Staubli VAL3: TEACH.pjx

--- TEACH.pjx ---
Parameters version=s7.7.1 stackSize=5000 millimeterUnit=true
Program file=AdjustTraj.pgx
Program file=Approach.pgx
Program file=Cut.pgx
Program file=GetListItems.pgx
Program file=GetProductMess.pgx
Program file=IdlePoint.pgx
Program file=IsPointOK.pgx
Program file=Leave.pgx
Program file=OnAction.pgx
Program file=OneWpMproChoose.pgx
Program file=Product.pgx
Program file=SetTrajPara.pgx
Program file=Simulate.pgx
Program file=SingleMove.pgx
Program file=start.pgx
Program file=stop.pgx
Program file=Teach2Tool.pgx
Program file=TeachAction.pgx
Program file=TeachAxis.pgx
Program file=TeachConfig.pgx
Program file=TeachFrame.pgx
Program file=TeachHome.pgx
Program file=TeachNewTraj.pgx
Program file=TeachOffset.pgx
Program file=TeachPreset.pgx
Program file=TeachProduct.pgx
Program file=TeachRecipe.pgx
Program file=TeachRemote.pgx
Program file=TeachSyncAxis.pgx
Program file=TeachTool.pgx
Program file=TrajScreen.pgx
Program file=WeldTraj.pgx
Program file=WorkPlaceChose.pgx
Data file=Teach.dtx
Library alias=TxtFile path=Disk://TxtFile/TxtFile.pjx
Library alias=DataBase path=Disk://DataBase/DataBase.pjx
Library alias=Kit path=Disk://Kit/Kit.pjx
Library alias=UI path=Disk://StaubliUI/StaubliUI.pjx
Library alias=Motion path=Disk://Motion/Motion.pjx
Library alias=IO path=Disk://IO/IO.pjx
Library alias=Algorith path=Disk://Algorith/Algorith.pjx
Library alias=CalTool path=Disk://StaubliCalTool7/StaubliCalTool7.pjx
Library alias=ExtAxis path=Disk://extAxisCan/extAxisCan.pjx autoload=false
Library alias=Custom path=Disk://Custom/Custom.pjx

--- TEACH.dtx ---
mdesc mNomSpeed
num nApproIndex
num nCutIndex
num nLeaveIndex
public num nPointType
string sSItem
public num nTrajIndex
public string sMess
num nCutMc
bool bPowerFlag
bool bFirstTeach
num nTeachAction
bool bSyc
public num n500Count
num nPartID
bool bSaveTxt
bool bCheckAxisSafte
num nCursonIndex
num nAxisSpeed

--- start.pgx ---
public program start()
begin














end

--- AdjustTraj.pgx ---
public program AdjustTraj(num x_nTrajIndex)
  local bool l_bRes
  local num l_nNum
begin


  //调图主界面，入口

  cls()

  call UI:Control_PanelMd("请等待，正在读取文件......")
  TxtFile:bStartRead=true
  DataBase:bStopPoll=true

  //删除临时文件
  if $fileExists("Disk://Txt/1.txt")
    $delete("Disk://Txt/1.txt")
  endIf

  if $fileExists("Disk://Txt/2.txt")
    $delete("Disk://Txt/2.txt")
  endIf

  if $fileExists("Disk://Txt/3.txt")
    $delete("Disk://Txt/3.txt")
  endIf

  if $fileExists("Disk://Txt/4.txt")
    $delete("Disk://Txt/4.txt")
  endIf




  call TxtFile:IsAdjustTraj("Disk://Txt/Recipe.txt",TxtFile:sProductName,x_nTrajIndex,x_nTrajIndex,l_bRes)
  call TxtFile:CloseFile()
  if !l_bRes
    DataBase:bStopPoll=false
    popUpMsg("文件读取出错!")
    return
  endIf


  //参数初始化
  bFirstTeach=true
  DataBase:bStopPoll=false
  //路径界面
  call TrajScreen()


end

--- APPROACH.pgx ---
public program Approach()
  local num l_nKey
  local bool l_bRes
  local string l_sProductName
  local jointRx l_jBuff
  local bool l_bCut
  local bool l_bMoveL
  local bool l_bFirst
  local trsf l_trTrsf
  local num l_nNum
  local num l_nAtPosition
begin
  //趋近点主界面
  //  $jogContext(TxtFile:tCfg,TxtFile:fArray,0)








  TxtFile:fArray.trsf={0,0,0,0,0,0}

  //2014.2.17  在哪个坐标系中运动
  if !DataBase:bWorldMove
    $jogContext(TxtFile:tCfg,TxtFile:fArray,0)
  else
    $jogContext(TxtFile:tCfg,world,0)
  endIf


  call IO:KeyDigtalIO(false,false,false,0,0)

  TxtFile:fArray.trsf={0,0,0,0,0,0}
  cls()
  while  nPointType==1
    l_nKey=getKey()
    switch l_nKey
      //上移
      case 261
        nApproIndex=max(nApproIndex-1,0)


      break

      //下移
      case 266
        nApproIndex=min(nApproIndex+1,size(TxtFile:pAppro)-1)

      break


      //向右
      //2015.08.10
      case 268
        nPointType=2
      break


      //插入
      case 271

        insert(TxtFile:pAppro[nApproIndex+1])
        insert(TxtFile:jAppro[nApproIndex+1])
        insert(TxtFile:bAppro[nApproIndex+1])
        insert(TxtFile:trAppro[nApproIndex+1])
        //外部轴
        insert(TxtFile:trApproAxis[nApproIndex+1])
        TxtFile:pAppro[nApproIndex+1]=TxtFile:pAppro[nApproIndex]
        TxtFile:jAppro[nApproIndex+1]=TxtFile:jAppro[nApproIndex]
        TxtFile:bAppro[nApproIndex+1]=TxtFile:bAppro[nApproIndex]
        TxtFile:trAppro[nApproIndex+1]=TxtFile:trAppro[nApproIndex]
        //外部轴
        TxtFile:trApproAxis[nApproIndex+1]=TxtFile:trApproAxis[nApproIndex]


        nApproIndex=nApproIndex+1
        TxtFile:trPointCount.x=size(TxtFile:pAppro)

        //2014.5.30
        //××××××××××××××××××××××
        if TxtFile:nSingleType!=20 and TxtFile:nSingleType!=9
          TxtFile:pAppro[nApproIndex]=here(TxtFile:tCfg,TxtFile:fArray)
          if TxtFile:fPofffset.trsf=={0,0,0,0,0,0} and TxtFile:fToffset.trsf=={0,0,0,0,0,0} and TxtFile:fArray.trsf=={0,0,0,0,0,0}
            TxtFile:jAppro[nApproIndex]=herej()
          else
            call Motion:Point2Joint(TxtFile:pAppro[nApproIndex], TxtFile:jAppro[nApproIndex],l_bRes)
            if !l_bRes
              popUpMsg("Joint数据转换出错")
            endIf
          endIf
        endIf

        //××××××××××××××××××××××××




      break


      //记录
      case 272
        TxtFile:fArray.trsf={0,0,0,0,0,0}
        //2015.08.10
        l_bRes=true
        //call UI:Control_YesNO("确定要记录吗?",l_bRes)

        if l_bRes
          TxtFile:pAppro[nApproIndex]=here(TxtFile:tCfg,TxtFile:fArray)
          if TxtFile:fPofffset.trsf=={0,0,0,0,0,0} and TxtFile:fToffset.trsf=={0,0,0,0,0,0} and TxtFile:fArray.trsf=={0,0,0,0,0,0}
            TxtFile:jAppro[nApproIndex]=herej()
          else
            call Motion:Point2Joint(TxtFile:pAppro[nApproIndex], TxtFile:jAppro[nApproIndex],l_bRes)
            if !l_bRes
              popUpMsg("Joint数据转换出错")
            endIf
          endIf

          //2014.07.28记录同步外部轴
          if TxtFile:nSingleType==20 or TxtFile:nSingleType==9
            call ExtAxis:RecordExtAxis(TxtFile:trApproAxis[nApproIndex],TxtFile:pAppro[nApproIndex].trsf,TxtFile:tCfg)
          endIf


        endIf
      break

      //参数
      case 273
        l_bMoveL=TxtFile:bAppro[nApproIndex]
        // call UI:Control_Para(TxtFile:trAppro[nApproIndex],TxtFile:bAppro[nApproIndex],false,0)
        call UI:Control_Para(TxtFile:trAppro,TxtFile:bAppro,false,TxtFile:nSingleType,nApproIndex,TxtFile:trApproAxis)
        //改变标志符
        if l_bMoveL!=TxtFile:bAppro[nApproIndex]
          //MOVEL
          if TxtFile:bAppro[nApproIndex]
            call Motion:Joint2Point(TxtFile:jAppro[nApproIndex],TxtFile:pAppro[nApproIndex])
          else
            //MOVEJ
            call Motion:Point2Joint(TxtFile:pAppro[nApproIndex], TxtFile:jAppro[nApproIndex],l_bRes)
            if !l_bRes
              popUpMsg("Joint数据转换出错")
            endIf
          endIf

          //2014.12.05记录同步外部轴
          if TxtFile:nSingleType==20 or TxtFile:nSingleType==9
            call ExtAxis:RecordExtAxis(TxtFile:trApproAxis[nApproIndex],TxtFile:pAppro[nApproIndex].trsf,TxtFile:tCfg)
          endIf


        endIf
      break

      //删除
      case 274
        if size(TxtFile:pAppro)==1
          popUpMsg("趋近点必须有一个")
        else
          call UI:Control_YesNO("确定要删除吗?",l_bRes)
          if l_bRes
            delete(TxtFile:pAppro[nApproIndex])
            delete(TxtFile:jAppro[nApproIndex])
            delete(TxtFile:bAppro[nApproIndex])
            delete(TxtFile:trAppro[nApproIndex])
            delete(TxtFile:trApproAxis[nApproIndex])
          endIf
        endIf
        TxtFile:trPointCount.x=size(TxtFile:pAppro)
      break


      //配置
      case 112,275
        call SetTrajPara()


      break

      //退出
      case 277
        call UI:Control_YesNO("确定要退出吗?",l_bRes)
        if l_bRes
          nPointType=-1
          return
        endIf
      break

      //上传
      case 278
        nPointType=2
      break

      //点位
      case 270
        if TxtFile:bAppro[nApproIndex]
          call UI:Control_Point(TxtFile:pAppro[nApproIndex] )
        else
          call UI:Control_Joint(TxtFile:jAppro[nApproIndex])
        endIf
        cls()
      break

      //****************************************
      //V
      //2014.12.02
      //外部PLC控制第七轴
      case 118
        if DataBase:bExtraContrAxis
          call UI:Control_YesNO("确定移动外部第七轴吗？",l_bRes)
          if l_bRes
            call UI:Control_PanelMd("外部第七轴正在运动....")
            resetMotion()
            call IO:ExtraContrAxis(TxtFile:trWorkplace.x,l_bRes)
            if !l_bRes
              popUpMsg("PLC控制外部轴数据错误,检查第七轴数据!")
              disablePower()
            endIf
          endIf
          cls()
        endIf
      break
      //******************************************




    endSwitch





    if (l_nKey<279  and l_nKey>=260)or l_nKey==112 or !l_bFirst or l_nKey==118
      l_bFirst=true
      call GetListItems()
      call UI:Form_PanelList("LasMAN3.6->示教路径","趋近点",sSItem,nApproIndex,"插入,记录,参数,删除,全局,,退出,继续")
      call UI:Control_Mess("类型:"+TxtFile:sTrajType[TxtFile:nSingleType],"趋近点个数:"+toString("",size(TxtFile:pAppro)))
      call SingleMove(1)



    endIf
    //2014.07.30
    //同步七八轴
    if (TxtFile:nSingleType==20 or TxtFile:nSingleType==9) and (TxtFile:bSync7Axis or TxtFile:bSync8Axis)
      call ExtAxis:RecordExtAxis(l_trTrsf,l_trTrsf,TxtFile:tCfg)

      gotoxy(1,12)
      put("七轴:"+toString(".3",l_trTrsf.x))
      if TxtFile:bSync8Axis
        gotoxy(20,12)
        put("八轴:"+toString(".3",l_trTrsf.y))
      endIf
    endIf
    //

    //为了表示到达位置
    //2015.08.10
    //2015.09.22
    //为整个列表进行修改

    if nApproIndex>10
      l_nAtPosition=nApproIndex-10
    else
      l_nAtPosition=0
    endIf

    for l_nNum=0 to min(size(TxtFile:bAppro)-1,10)
      gotoxy(22,min(l_nNum+1,10))
      setTextMode(sel((l_nAtPosition+l_nNum)==nApproIndex,1,0))


      if TxtFile:bAppro[l_nAtPosition+l_nNum]
        if distance(TxtFile:pAppro[l_nAtPosition+l_nNum],here(TxtFile:tFileTool,TxtFile:fArray))<0.1
          put("@")
        else
          put("│")
        endIf

      else
        if distance(jointToPoint(TxtFile:tFileTool,TxtFile:fArray,herej()),jointToPoint(TxtFile:tFileTool,TxtFile:fArray,TxtFile:jAppro[l_nAtPosition+l_nNum]))<0.1
          put("@")
        else
          put("│")
        endIf
      endIf
    endFor

    //*************************

    delay(0)

  endWhile



end

--- CUT.pgx ---
public program Cut()
  local num l_nKey
  local bool l_bRes
  local string l_sProductName
  local string l_sBottom
  local bool l_bCut
  local num l_nSaveTime
  local frame l_trOffset
  local num l_nTo[5]
  local num l_nFrom[5]
  local num l_nNum
  local bool l_bFirst
  local num l_nSpeed[2]
  local string l_sTtile
  local bool l_bBatPara[5]
  local num l_nBatPara[5]
  local num l_nFromTo[2]
  local trsf l_trTrsf
  local num l_nAtPosition
begin
  //切割点主界面
  //参数初始化
  // call IO:Follow(false)
  call IO:SafteyIO()
  TxtFile:fArray.trsf={0,0,0,0,0,0}


  //2014.2.17  在哪个坐标系中运动
  if !DataBase:bWorldMove
    $jogContext(TxtFile:tCfg,TxtFile:fArray,0)
  else
    $jogContext(TxtFile:tCfg,world,0)
  endIf

  //2014.2.18 区分焊接与切割
  if TxtFile:bWeldEnable
    l_sTtile="焊接点"
  else
    l_sTtile="切割点"
  endIf



  nPartID=1
  if TxtFile:trPointCount.y>500
    DataBase:bStopPoll=true
    call TxtFile:ReadPartTraj(nPartID,l_bRes)
  endIf
  DataBase:bStopPoll=false
  nCutMc=0
  l_nSaveTime=0
  n500Count=0

  if TxtFile:nSingleType!=10 and TxtFile:nSingleType!=20 and TxtFile:nSingleType!=9

    for l_nKey=0 to size(TxtFile:pCut)-1
      TxtFile:bMoveC[l_nKey]=false
    endFor
  endIf

  //界面
  call GetListItems()
  if TxtFile:nSingleType==10 or TxtFile:nSingleType==20
    l_sBottom="插入,记录,参数,删除,全局,偏差,返回,继续"
  else
    l_sBottom=",记录,参数,,全局,偏差,返回,继续"
  endIf


  //界面初始化
  resetMotion()
  cls()


  //循环
  while  nPointType==2
    DataBase:bStopPoll=false
    TxtFile:fArray.trsf={0,0,0,0,0,0}
    l_nKey=getKey()
    switch l_nKey

      //配置
      case 112,275
        call SetTrajPara()


      break

      //步进打开
      case 122
        //Z
        // if TxtFile:bStepMove
        TxtFile:nStepLength=max(0,TxtFile:nStepLength)
        call UI:Control_YesNO("确定使用步进"+toString(".1",TxtFile:nStepLength)+"毫米模式吗?",l_bRes)
        if l_bRes
          TxtFile:fArray.trsf={0,0,0,0,0,0}
          $jogContext(TxtFile:tCfg,TxtFile:fArray,TxtFile:nStepLength)
        endIf
        //  endIf
      break


      //步进关
      case 90

        TxtFile:fArray.trsf={0,0,0,0,0,0}
        $jogContext(TxtFile:tCfg,TxtFile:fArray,0)
        popUpMsg("不使用步进模式")
      break


      //快捷设置
      case 113
        //Q
        call UI:Control_YesNO("确定要使用快捷参数吗?",l_bRes)
        if l_bRes
          //工艺
          TxtFile:trCut[nCutIndex].z=TxtFile:trCorner.x
          //速度
          TxtFile:trCut[nCutIndex].z=TxtFile:trCorner.z
          //加速度
          TxtFile:trCut[nCutIndex].rx=TxtFile:trCorner.rx
          //blend
          TxtFile:trCut[nCutIndex].ry=TxtFile:trCorner.ry
        endIf


      break

      //向上
      case 261
        nCursonIndex=nCutIndex
        nCutMc=0
        nCutIndex=nCutIndex-1
        if nCutIndex<0
          nCutIndex=size(TxtFile:pCut)-1
        endIf
        nCutIndex=max(nCutIndex,0)


      break

      //向下
      case 266
        nCursonIndex=nCutIndex
        nCutMc=0
        nCutIndex=nCutIndex+1
        if nCutIndex>=size(TxtFile:pCut)
          nCutIndex=0
        endIf
        nCutIndex=min(nCutIndex,size(TxtFile:pCut)-1)
      break

      //向左
      case 264
        //2015.08.16
        if  TxtFile:bMoveC[nCutIndex]
          nCutMc=max(0,nCutMc-1)
        else
          nPointType=1
        endIf
      break

      //向右
      case 268
        if  TxtFile:bMoveC[nCutIndex]
          nCutMc=min(2,nCutMc+1)
        else
          nPointType=3
        endIf


      break
      //点位
      case 270
        if  TxtFile:bMoveC[nCutIndex] and nCutMc==1
          call UI:Control_Point(TxtFile:pMoveC[nCutIndex])

        else
          if TxtFile:bMoveC[nCutIndex] and nCutMc==2 or !TxtFile:bMoveC[nCutIndex]
            call UI:Control_Point(TxtFile:pCut[nCutIndex])
          endIf
        endIf


      break


      //插入
      case 271
        if TxtFile:nSingleType==10 or TxtFile:nSingleType==20
          if  (!insert(TxtFile:pCut[nCutIndex+1])) or (!insert(TxtFile:bMoveC[nCutIndex+1])) or (!insert(TxtFile:pMoveC[nCutIndex+1])) or (!insert(TxtFile:trCut[nCutIndex+1]))  or (!insert(TxtFile:trCutAxis[nCutIndex+1]))
            popUpMsg("插入失败")
          else
            TxtFile:pCut[nCutIndex+1]=TxtFile:pCut[nCutIndex]
            TxtFile:bMoveC[nCutIndex+1]=TxtFile:bMoveC[nCutIndex]
            TxtFile:pMoveC[nCutIndex+1]=TxtFile:pMoveC[nCutIndex]
            TxtFile:trCut[nCutIndex+1]=TxtFile:trCut[nCutIndex]
            TxtFile:trCutAxis[nCutIndex+1]=TxtFile:trCutAxis[nCutIndex]
            nCutIndex=nCutIndex+1

            //2014.05.30
            if TxtFile:nSingleType!=20 and TxtFile:nSingleType!=9
              TxtFile:pMoveC[nCutIndex]=here(TxtFile:tCfg,TxtFile:fArray)
              TxtFile:pCut[nCutIndex]=here(TxtFile:tCfg,TxtFile:fArray)
            else
              //2015.03.21
              call ExtAxis:RecordExtAxis(TxtFile:trCutAxis[nCutIndex],TxtFile:pMoveC[nCutIndex].trsf,TxtFile:tCfg)
              call ExtAxis:RecordExtAxis(TxtFile:trCutAxis[nCutIndex],TxtFile:pCut[nCutIndex].trsf,TxtFile:tCfg)

            endIf

            //×××××××××××××××××××××××××××××××8


          endIf

        endIf
        //        TxtFile:trPointCount.y=size(TxtFile:pCut)

      break

      //记录
      case 272
        if !((TxtFile:nSingleType==10 or TxtFile:nSingleType==20)and TxtFile:bMoveC[nCutIndex] and nCutMc==0)
          //2015.08.10
          l_bRes=true
          // call UI:Control_YesNO("确定要记录吗?",l_bRes)
          if l_bRes
            //2014.12.08
            //为同步轴进行修改
            if TxtFile:bMoveC[nCutIndex]
              if nCutMc==1
                TxtFile:pMoveC[nCutIndex]=here(TxtFile:tCfg,TxtFile:fArray)
              else
                TxtFile:pCut[nCutIndex]=here(TxtFile:tCfg,TxtFile:fArray)
              endIf
            else
              TxtFile:pMoveC[nCutIndex]=TxtFile:pCut[nCutIndex]=here(TxtFile:tCfg,TxtFile:fArray)
            endIf
            //2014.07.28记录同步外部轴
            if TxtFile:nSingleType==20
              if TxtFile:bMoveC[nCutIndex] and nCutMc==1

                call ExtAxis:RecordExtAxis(TxtFile:trCutAxis[nCutIndex],TxtFile:pMoveC[nCutIndex].trsf,TxtFile:tCfg)
              else
                call ExtAxis:RecordExtAxis(TxtFile:trCutAxis[nCutIndex],TxtFile:pCut[nCutIndex].trsf,TxtFile:tCfg)
              endIf
            endIf
          endIf
        endIf






      break

      //参数
      case 273
        //  call UI:Form_4jHome()
        call UI:Control_Para(TxtFile:trCut,TxtFile:bMoveC,true,TxtFile:nSingleType,nCutIndex,TxtFile:trCutAxis)
        //强制赋值为false
        if (TxtFile:nSingleType!=10 and TxtFile:nSingleType!=20)
          TxtFile:bMoveC[nCutIndex]=false
        endIf

        if TxtFile:trPointCount.x<500
          TxtFile:bMoveC[0]=false
        endIf


      break

      //删除
      case 274
        if TxtFile:nSingleType==10 or TxtFile:nSingleType==20
          if size(TxtFile:pCut)==1
            popUpMsg(l_sTtile+"必须有一个")
          else
            call UI:Control_YesNO("确定要删除吗?",l_bRes)
            if l_bRes
              //              if  !delete(TxtFile:pCut[nCutIndex]) or !delete(TxtFile:pMoveC[nCutIndex]) or !delete(TxtFile:bMoveC[nCutIndex]) or !delete(TxtFile:trCut[nCutIndex])
              //                popUpMsg("删除失败")
              //              endIf
              delete(TxtFile:pCut[nCutIndex])
              delete(TxtFile:pMoveC[nCutIndex])
              delete(TxtFile:bMoveC[nCutIndex])
              delete(TxtFile:trCut[nCutIndex])
              delete(TxtFile:trCutAxis[nCutIndex])

            endIf
          endIf
        endIf
        //        if TxtFile:trPointCount.y<500
        //            TxtFile:trPointCount.y=size(TxtFile:pCut)
        //        endIf
        nCutIndex=min(size(TxtFile:pCut)-1,nCutIndex)

      break

      //对齐
      case 100
        call Kit:Align(TxtFile:tCfg)

      break

      //偏差
      case 276
        call UI:Control_YesNO("确定要示教偏差吗?",l_bRes)
        if l_bRes
          call TeachOffset(TxtFile:fToffset)

        endIf
      break

      //返回
      case 277
        if  TxtFile:trPointCount.y>500
          //          call UI:Control_YesNO("切割点是否需要进行局部保存",l_bRes)
          //          if l_bRes
          DataBase:bStopPoll=true
          call TxtFile:SavePartTraj(nPartID,l_bRes)
          DataBase:bStopPoll=false
          if l_bRes
            //popUpMsg("保存成功")
            TxtFile:nPartTrajCount[nPartID]=size(TxtFile:pCut)
          else
            popUpMsg("局部切割路径保存失败")
          endIf
          //          endIf
        endIf


        if bFirstTeach==false or TxtFile:trPointCount.y<=500 or (TxtFile:nSingleType!=10 and TxtFile:nSingleType!=20) or nPartID<=1
          nPointType=1
        else
          nPartID=nPartID-1
          DataBase:bStopPoll=true
          call TxtFile:ReadPartTraj(nPartID,l_bRes)
          DataBase:bStopPoll=false
          if !l_bRes
            popUpMsg("读取文件出错")
          endIf
        endIf
      break


      //继续
      case 278
        //        if bFirstTeach==false or TxtFile:trPointCount.y<=500 or TxtFile:nSingleType!=10 or nPartID*500>TxtFile:trPointCount.y
        if  TxtFile:trPointCount.y>500 or size(TxtFile:pCut)>500
          //          call UI:Control_YesNO("切割点是否需要进行局部保存",l_bRes)
          //          if l_bRes
          DataBase:bStopPoll=true
          call TxtFile:SavePartTraj(nPartID,l_bRes)
          DataBase:bStopPoll=false
          if l_bRes
            //popUpMsg("保存成功")
            TxtFile:nPartTrajCount[nPartID]=size(TxtFile:pCut)
          else
            popUpMsg("局部路切割径保存失败")
          endIf
          //          endIf
        endIf


        if nPartID*500>TxtFile:trPointCount.y or TxtFile:trPointCount.y<=500
          nPointType=3
        else


          nPartID=nPartID+1
          DataBase:bStopPoll=true
          call TxtFile:ReadPartTraj(nPartID,l_bRes)
          DataBase:bStopPoll=false
          if !l_bRes
            popUpMsg("读取文件出错")
          else
            nCutIndex=0
          endIf
        endIf
      break

      //示教局部偏差
      case 119
        call UI:Control_YesNO("确定要示教局部偏差吗?",l_bRes)
        link(l_trOffset,TxtFile:fToffset)
        if l_bRes
          l_trOffset.trsf={0,0,0,0,0,0}
          call TeachOffset(l_trOffset)
          if l_trOffset.trsf!={0,0,0,0,0,0}
            l_nFromTo[0]=l_nFromTo[1]=0
            call UI:Control_Loffset(l_nFromTo[0],l_nFromTo[1])
            if l_nFromTo[0]!=0 and l_nFromTo[1]!=0
              l_nFromTo[0]=max(0,l_nFromTo[0])
              l_nFromTo[1]=min(l_nFromTo[1],size(TxtFile:pCut))
              for l_nNum=l_nFromTo[0] to l_nFromTo[1]
                TxtFile:pCut[l_nNum].trsf=l_trOffset.trsf*TxtFile:pCut[l_nNum].trsf
                TxtFile:pMoveC[l_nNum].trsf=l_trOffset.trsf*TxtFile:pMoveC[l_nNum].trsf

              endFor
              popUpMsg("偏差已修正,请模拟")
            endIf
          endIf
        endIf




      break


      //局部模拟
      case 115
        //数据预设
        DataBase:nPartMove[2]=nCutIndex
        DataBase:nPartMove[0]=nCutIndex+1
        DataBase:nPartMove[1]=size(TxtFile:pCut)
        if TxtFile:nSingleType!=10 or size(TxtFile:pCut)<=1
          popUpMsg("规则图形与点数小于1不能进行局部模拟")

        else

          call UI:Control_YesNO("确定要进行局部模拟吗",l_bRes)
          if l_bRes
            call UI:Control_PatMove(DataBase:nPartMove[0],DataBase:nPartMove[1])
            //输入数据合法处理
            DataBase:nPartMove[0]=roundDown(DataBase:nPartMove[0])
            DataBase:nPartMove[1]=roundDown(DataBase:nPartMove[1])
            DataBase:nPartMove[0]=min(size(TxtFile:pCut)-1,max(1,DataBase:nPartMove[0]))
            DataBase:nPartMove[1]=min(size(TxtFile:pCut),max(DataBase:nPartMove[0]+1,DataBase:nPartMove[1]))
            TxtFile:nReadCutCount=DataBase:nPartMove[1]-DataBase:nPartMove[0]+1
            call Simulate(-2)
            call IO:SafteyIO()
            call UI:Control_PanelMd("模拟结束")
            delay(2)
            cls()
          endIf

        endIf
        DataBase:nPointType=2
        nPointType=2
        nCutIndex=DataBase:nPartMove[2]
      break


      //      //局部保存
      //      case 120
      //
      //        if TxtFile:nSingleType==10
      //          call UI:Control_YesNO("确定要局部保存吗?",l_bRes)
      //          if l_bRes
      //            call TxtFile:SavePartTraj(nPartID,l_bRes)
      //            if l_bRes
      //              popUpMsg("保存成功")
      //              TxtFile:nPartTrajCount[nPartID]=size(TxtFile:pCut)
      //            else
      //              popUpMsg("保存失败")
      //            endIf
      //
      //          endIf
      //        endIf
      //
      //
      //
      //
      //
      //      break


      //批处理参数
      case 101
        call UI:Control_YesNO("确定要批处理参数吗?",l_bRes)
        if l_bRes
          //          l_nSpeed[0]=l_nSpeed[1]=0
          //          l_nFromTo[0]=1
          //          l_nFromTo[1]=size(TxtFile:pCut)
          //          call UI:Control_BatSpd(l_nFromTo[0],l_nFromTo[1],l_nSpeed[0],l_nSpeed[1])
          //l_nFrom=resize(size(TxtFile:pCut))
          call UI:Control_BatPara(size(TxtFile:pCut),l_nFrom,l_nTo,l_nBatPara,l_bBatPara)
          if l_bRes
            //          if l_nFromTo[0]>0 and l_nFromTo>0 and l_nSpeed[0]>=0 and l_nSpeed[1]>=0 and l_nFromTo[1]>=l_nFromTo[0]


            for l_nSpeed[1]=0 to 4
              if l_bBatPara[l_nSpeed[1]]
                l_nFrom[l_nSpeed[1]]=max(0,l_nFrom[l_nSpeed[1]])
                l_nTo[l_nSpeed[1]]=min(l_nTo[l_nSpeed[1]],size(TxtFile:pCut))
                l_nSpeed[0]=l_nBatPara[l_nSpeed[1]]
                for l_nNum= l_nFrom[l_nSpeed[1]] to l_nTo[l_nSpeed[1]]
                  //              TxtFile:trCut[l_nNum-1].z=l_nSpeed[0]
                  //              TxtFile:trCut[l_nNum-1].rx=l_nSpeed[1]
                  switch l_nSpeed[1]
                    case 0
                      TxtFile:trCut[l_nNum-1].z=l_nSpeed[0]
                    break

                    case 1
                      TxtFile:trCut[l_nNum-1].rx=l_nSpeed[0]
                    break
                    case 2
                      TxtFile:trCut[l_nNum-1].ry=l_nSpeed[0]
                    break
                    case 3
                      TxtFile:trCut[l_nNum-1].x=l_nSpeed[0]
                    break
                    case 4
                      TxtFile:trCut[l_nNum-1].y=l_nSpeed[0]
                    break

                  endSwitch

                endFor
              endIf
            endFor
            if l_bBatPara[0] or l_bBatPara[1] or l_bBatPara[2] or l_bBatPara[3] or l_bBatPara[4]
              popUpMsg("参数已修改")
            endIf
          endIf
        endIf

      break




      //x 修改工艺
      case 120
        call UI:Control_CPreset(TxtFile:nPreset,TxtFile:trCut,size(TxtFile:trCut),nCutIndex,TxtFile:trCutAxis)

        cls()
      break

      //      //批处理工艺
      //      case 99
      //        call UI:Control_YesNO("确定要批处理工艺吗?",l_bRes)
      //        if l_bRes
      //          l_nSpeed[0]=l_nSpeed[1]=0
      //          l_nFromTo[0]=1
      //          l_nFromTo[1]=size(TxtFile:pCut)
      //          call UI:Control_BatPrt(l_nFromTo[0],l_nFromTo[1],l_nSpeed[0])
      //          if l_nFromTo[0]>0  and l_nSpeed[0]>0  and l_nFromTo[1]>=l_nFromTo[0]
      //            l_nFromTo[0]=max(0,l_nFromTo[0])
      //            l_nFromTo[1]=min(l_nFromTo[1],size(TxtFile:pCut))
      //            for l_nNum=l_nFromTo[0] to l_nFromTo[1]
      //              TxtFile:trCut[l_nNum-1].x=l_nSpeed[0]
      //            endFor
      //            popUpMsg("工艺已修改")
      //          endIf
      //        endIf
      //
      //
      //      break

    endSwitch
    n500Count=max(nPartID-1,0)

    //界面刷新
    if (l_nKey>=97 and l_nKey<279) or !l_bFirst or l_nKey==120

      //机械手臂移动
      if l_nKey==97 or l_nKey==122
      else
        call SingleMove(2)
      endIf

      //界面
      l_bFirst=true
      call GetListItems()
      call UI:Form_PanelList("LasMAN3.6->示教路径",l_sTtile,sSItem,nCutIndex,l_sBottom)
      call UI:Control_LeftCut(2)
      call UI:Control_Mess("类型:"+TxtFile:sTrajType[TxtFile:nSingleType],l_sTtile+"个数:"+toString("",size(TxtFile:pCut)))
      if TxtFile:bMoveC[nCutIndex]
        call UI:Control_MCShow(nCutIndex,nCutMc)
      endIf


      //


    endIf

    //2014.11.28
    //强制第一个点是MOVEL
    if TxtFile:trPointCount.y<500
      TxtFile:bMoveC[0]=false
    endIf






    //2014.7.30
    //同步七八轴
    if TxtFile:nSingleType==20 and (TxtFile:bSync7Axis or TxtFile:bSync8Axis)
      call ExtAxis:RecordExtAxis(l_trTrsf,l_trTrsf,TxtFile:tCfg)
      gotoxy(0,12)
      put("七轴:"+toString(".3",l_trTrsf.x))
      if TxtFile:bSync8Axis
        gotoxy(20,12)
        put("八轴:"+toString(".3",l_trTrsf.y))
      endIf
    endIf



    //根据值来进行判断
    //call IO:Follow(true)

    //示教操作20分，则自动保存
    if clock()-l_nSaveTime>1200
      l_nSaveTime=clock()
      //  taskCreate "AutoSave",100,TxtFile:SaveAutoTraj()
    endIf



    //为了表示到达位置
    //2015.08.10
    //2015.09.22
    //为整个列表进行修改

    if nCutIndex>10
      l_nAtPosition=nCutIndex-10
    else
      l_nAtPosition=0
    endIf

    for l_nNum=0 to min(size(TxtFile:bMoveC)-1,10)
      gotoxy(22,min(l_nNum+1,10))
      setTextMode(sel((l_nAtPosition+l_nNum)==nCutIndex,1,0))

      //2015.8.25
      //MOVEC添加到位
      if TxtFile:bMoveC[l_nAtPosition+l_nNum]==false or (TxtFile:bMoveC[l_nAtPosition+l_nNum] and nCutMc!=1)
        if distance(TxtFile:pCut[l_nAtPosition+l_nNum],here(TxtFile:tFileTool,TxtFile:fArray))<0.1
          put("@")
        else
          put("│")
        endIf
      else

        if distance(TxtFile:pMoveC[l_nAtPosition+l_nNum],here(TxtFile:tFileTool,TxtFile:fArray))<0.1
          put("@")
        else
          put("│")
        endIf
      endIf
    endFor


    //*************************




    delay(0)

  endWhile



end

--- GetListItems.pgx ---
program GetListItems()
  local num l_nNum
  local num l_nCount
begin
  //获取选项框中列表
  if DataBase:nInterfaceType!=13
    switch nPointType
      case 1
        resize(sSItem,1,size(TxtFile:pAppro,1))
        for l_nNum=0 to size(TxtFile:bAppro,1)-1
          if TxtFile:bAppro[l_nNum]
            sSItem[l_nNum]=toString("",l_nNum+1)+"."+"MoveL"

          else
            sSItem[l_nNum]=toString("",l_nNum+1)+"."+"MoveJ"
          endIf

        endFor

      break


      case 2
        resize(sSItem,1,size(TxtFile:pCut,1))
        for l_nNum=0 to size(TxtFile:bMoveC,1)-1
          if TxtFile:bMoveC[l_nNum]
            sSItem[l_nNum]=toString("",l_nNum+1+500*n500Count)+"."+"MoveC 1  2"

          else
            sSItem[l_nNum]=toString("",l_nNum+1+500*n500Count)+"."+"MoveL"
          endIf

          //焊接的话，把动作放在外面
          if TxtFile:bWeldEnable and TxtFile:trWorkplace.z==1

            sSItem[l_nNum]=sSItem[l_nNum]+"_"+toString("",TxtFile:trCut[l_nNum].y)
          endIf


        endFor
        if  size(TxtFile:pCut)==1 and (TxtFile:nSingleType==12 or TxtFile:nSingleType==2 or TxtFile:nSingleType==23)
          sSItem[0]="1.圆心点"
        else

          if TxtFile:nSingleType!=10 and TxtFile:nSingleType!=20 and size(TxtFile:pCut)==3
            //            sSItem[0]="1.第一点(原点)"
            //            sSItem[1]="2.第二点(X轴)"
            //            sSItem[2]="3.第三点(Y轴)"
            sSItem[0]="1.第一点"
            sSItem[1]="2.第二点"
            sSItem[2]="3.第三点"
          endIf
        endIf

      break

      case 3
        resize(sSItem,1,size(TxtFile:pLeave,1))
        for l_nNum=0 to size(TxtFile:bLeave,1)-1
          if TxtFile:bLeave[l_nNum]
            sSItem[l_nNum]=toString("",l_nNum+1)+"."+"MoveL"

          else
            sSItem[l_nNum]=toString("",l_nNum+1)+"."+"MoveJ"
          endIf

        endFor

      break




    endSwitch

  else
    switch DataBase:nPointType
      case 1
        l_nCount=TxtFile:trPointCount.x
      break

      case 2
        l_nCount=TxtFile:trPointCount.y
      break
      case 3
        l_nCount=TxtFile:trPointCount.z
      break
      default
        l_nCount=0
      break
    endSwitch
    sSItem[0]="---产品信息---"
    sSItem[1]="               "
    sSItem[2]="工位号:"+toString("",DataBase:nWorkPlaceIndex)+"->"+toString("",DataBase:nWorkPlaceCount)
    sSItem[3]="产品名:"+DataBase:sProductName[max(1,DataBase:nWorkPlaceIndex)]
    sSItem[4]="路径号:"+toString("",TxtFile:nReadTrajIndex)+"->"+toString("",TxtFile:nTotalTraj)
    sSItem[5]="点数号:"
    switch DataBase:nPointType
      case 1
        sSItem[5]=sSItem[5]+"趋"
      break
      case 2
        if !TxtFile:bWeldEnable
          sSItem[5]=sSItem[5]+"切"
        else
          sSItem[5]=sSItem[5]+"焊"
        endIf
      break

      case 3
        sSItem[5]=sSItem[5]+"离"
      break


    endSwitch

    sSItem[5]=sSItem[5]+toString(".1",DataBase:nID)+"->"+toString("",l_nCount)

    sSItem[6]="周期号:"+toString("",DataBase:nCycleIndex)+"->"+toString("",DataBase:nCycleCount)
    sSItem[7]="周期时间(秒):"+toString(".1",DataBase:nCycleTime)
    sSItem[8]="速度(m/min):"+toString(".2",DataBase:nRobotSpeed*60/1000)
    sSItem[9]="生产个数:"+toString("",DataBase:nProductCount)
    sSItem[10]="按钮触发:"
    if TxtFile:bMoreProd1Wp
      sSItem[10]=sSItem[10]+"同工多产"
    else
      switch DataBase:nCycleMode
        case 0
          sSItem[10]=sSItem[10]+"单工位"
        break

        case 1
          sSItem[10]=sSItem[10]+"单周期"
        break

        case 2
          sSItem[10]=sSItem[10]+"多周期"
        break
        case 3
          sSItem[10]=sSItem[10]+"无需触发"
        break

        case 4
          sSItem[10]=sSItem[10]+"排队("+toString("",DataBase:nWorkPlaceButto)+")"
        break
        case 5
          sSItem[10]=sSItem[10]+"自定义"
        break

      endSwitch


    endIf

    if TxtFile:bWeldEnable

      sSItem[11]="阵列:"+toString("",DataBase:nArrayX)+"->"+toString("",DataBase:nArrayY)+"->"+toString("",DataBase:nArrayZ)
    else
      sSItem[11]=""
    endIf


  endIf


end

--- GetProductMess.pgx ---
program GetProductMess(string x_sMess)
  local num l_nNum
begin
  //生产信息列表
  //专为生产界面


  sMess[0]="---生产日志---"
  sSItem[1]="               "
  if sMess[2]!=x_sMess


    for l_nNum=10 to 3 step -1
      sMess[l_nNum]=sMess[l_nNum-1]
    endFor
    sMess[2]=x_sMess
  endIf
end

--- IdlePoint.pgx ---
public program IdlePoint()
  local num l_nKey
  local bool l_bRes
  local string l_sProductName
  local jointRx l_jJBuff
  local bool l_bCut
  local bool l_bMoveL
  local num l_nNum
  local num l_nApproCount
  local bool l_bFirst
  local trsf l_trTrsf
  local num l_nIndex
begin


  //2015.2.12
  DataBase:bMoveTask=false
  call IO:KeyDigtalIO(false,false,false,0,0)
  TxtFile:nWeldActionId=0
  TxtFile:fArray.trsf={0,0,0,0,0,0}
  //2014.2.17  在哪个坐标系中运动
  if !DataBase:bWorldMove
    $jogContext(TxtFile:tCfg,TxtFile:fArray,0)
  else
    $jogContext(TxtFile:tCfg,world,0)
  endIf
  resize(sSItem,1,3)
  TxtFile:nTrajDelay[0]=TxtFile:nTrajDelay[1]=0
  TxtFile:trWorkplace.rz=-1

  //第一次示教,是否需要回退点
  if bFirstTeach==false
    bFirstTeach=true

    l_nApproCount=1
    resize(TxtFile:pLeave,1,l_nApproCount)
    resize(TxtFile:jLeave,1,l_nApproCount)
    resize(TxtFile:bLeave,1,l_nApproCount)
    resize(TxtFile:trLeave,1,l_nApproCount)
    resize(TxtFile:trLeaveAxis,1,l_nApproCount)

    resize(TxtFile:pAppro,1,l_nApproCount)
    resize(TxtFile:jAppro,1,l_nApproCount)
    resize(TxtFile:bAppro,1,l_nApproCount)
    resize(TxtFile:trAppro,1,l_nApproCount)
    resize(TxtFile:trApproAxis,1,l_nApproCount)

    resize(TxtFile:pCut,1,l_nApproCount)
    resize(TxtFile:pMoveC,1,l_nApproCount)
    resize(TxtFile:bMoveC,1,l_nApproCount)
    resize(TxtFile:trCut,1,l_nApproCount)
    resize(TxtFile:trCutAxis,1,l_nApproCount)


    //2015.04.21
    call ExtAxis:RecordExtAxis(TxtFile:trCutAxis[0],TxtFile:pMoveC[0].trsf,TxtFile:tCfg)
    call ExtAxis:RecordExtAxis(TxtFile:trCutAxis[0],TxtFile:pCut[0].trsf,TxtFile:tCfg)
    call ExtAxis:RecordExtAxis(TxtFile:trApproAxis[0],TxtFile:pAppro[0].trsf,TxtFile:tCfg)
    call ExtAxis:RecordExtAxis(TxtFile:trLeaveAxis[0],TxtFile:pLeave[0].trsf,TxtFile:tCfg)
    //    TxtFile:jAppro[0]=herej()
    call ExtAxis:RecordJoint(TxtFile:jAppro[0],TxtFile:trApproAxis[0])

    if l_nApproCount>1
      for l_nNum=0 to l_nApproCount-1
        TxtFile:bLeave[l_nNum]=TxtFile:bAppro[l_nApproCount-1-l_nNum]=false
        TxtFile:jLeave[l_nNum]=TxtFile:jAppro[l_nApproCount-1-l_nNum]
        TxtFile:pLeave[l_nNum]=TxtFile:pAppro[l_nApproCount-1-l_nNum]
        TxtFile:trLeave[l_nNum]=TxtFile:trAppro[l_nApproCount-1-l_nNum]

        TxtFile:trLeaveAxis[l_nNum]=TxtFile:trApproAxis[l_nApproCount-1-l_nNum]

      endFor
    endIf


  endIf







  TxtFile:trPointCount.z=size(TxtFile:pLeave)

  //界面初始化
  //  nPointType=3
  cls()
  while  true
    l_nKey=getKey()
    DataBase:bMoveTask=false
    TxtFile:nWeldActionId=0
    switch l_nKey

      //      //配置
      //      case 112
      //        call SetTrajPara()
      //
      //      break



      case 261
        l_nIndex=max(l_nIndex-1,0)


      break


      case 266
        l_nIndex=min(l_nIndex+1,2)


      break


      //      //插入
      //      case 271
      //
      //        insert(TxtFile:pLeave[nLeaveIndex+1])
      //        insert(TxtFile:jLeave[nLeaveIndex+1])
      //        insert(TxtFile:bLeave[nLeaveIndex+1])
      //        insert(TxtFile:trLeave[nLeaveIndex+1])
      //        insert(TxtFile:trLeaveAxis[nLeaveIndex+1])
      //
      //        TxtFile:pLeave[nLeaveIndex+1]=TxtFile:pLeave[nLeaveIndex]
      //        TxtFile:jLeave[nLeaveIndex+1]=TxtFile:jLeave[nLeaveIndex]
      //        TxtFile:bLeave[nLeaveIndex+1]=TxtFile:bLeave[nLeaveIndex]
      //        TxtFile:trLeave[nLeaveIndex+1]=TxtFile:trLeave[nLeaveIndex]
      //        TxtFile:trLeaveAxis[nLeaveIndex+1]=TxtFile:trLeaveAxis[nLeaveIndex]
      //        nLeaveIndex=nLeaveIndex+1
      //
      //        TxtFile:trPointCount.z=size(TxtFile:pLeave)
      //        //2014.05.30
      //        //××××××××××××××××××××××××××××××××××××××8
      //        if TxtFile:nSingleType!=20
      //          TxtFile:pLeave[nLeaveIndex]=here(TxtFile:tCfg,TxtFile:fArray)
      //          if TxtFile:fPofffset.trsf=={0,0,0,0,0,0} and TxtFile:fToffset.trsf=={0,0,0,0,0,0}
      //            TxtFile:jLeave[nLeaveIndex]=herej()
      //          else
      //            call Motion:Point2Joint(TxtFile:pLeave[nLeaveIndex], TxtFile:jLeave[nLeaveIndex],l_bRes)
      //            if !l_bRes
      //              popUpMsg("Joint数据转换出错")
      //            endIf
      //          endIf
      //        endIf
      //
      //        //×××××××××××××××××××××××××××××××××××××××××
      //
      //
      //
      //
      //
      //      break
      //

      //记录
      case 272
        TxtFile:fArray.trsf={0,0,0,0,0,0}
        call UI:Control_YesNO("确定要记录吗?",l_bRes)
        if l_bRes
          //          TxtFile:pLeave[nLeaveIndex]=here(TxtFile:tCfg,TxtFile:fArray)
          //          if TxtFile:fPofffset.trsf=={0,0,0,0,0,0} and TxtFile:fToffset.trsf=={0,0,0,0,0,0}
          //            TxtFile:jLeave[nLeaveIndex]=herej()
          //          else
          //            call Motion:Point2Joint(TxtFile:pLeave[nLeaveIndex], TxtFile:jLeave[nLeaveIndex],l_bRes)
          //            if !l_bRes
          //              popUpMsg("Joint数据转换出错")
          //            endIf
          //          endIf
          //          //2014.07.28记录同步外部轴
          //          if TxtFile:nSingleType==20
          //            call ExtAxis:RecordExtAxis(TxtFile:trLeaveAxis[nLeaveIndex],TxtFile:pLeave[nLeaveIndex].trsf,TxtFile:tCfg)
          //          endIf

          switch l_nIndex

            case 0
              TxtFile:pAppro[0]=here(TxtFile:tCfg,TxtFile:fArray)
              if TxtFile:fPofffset.trsf=={0,0,0,0,0,0} and TxtFile:fToffset.trsf=={0,0,0,0,0,0} and TxtFile:fArray.trsf=={0,0,0,0,0,0}
                TxtFile:jAppro[0]=herej()
              else
                call Motion:Point2Joint(TxtFile:pAppro[0], TxtFile:jAppro[0],l_bRes)
                if !l_bRes
                  popUpMsg("Joint数据转换出错")
                endIf
              endIf

              call ExtAxis:RecordExtAxis(TxtFile:trApproAxis[0],TxtFile:pAppro[0].trsf,TxtFile:tCfg)

            break

            case 1
              TxtFile:pCut[0]=here(TxtFile:tCfg,TxtFile:fArray)
              call ExtAxis:RecordExtAxis(TxtFile:trCutAxis[0],TxtFile:pCut[0].trsf,TxtFile:tCfg)
              call ExtAxis:RecordExtAxis(TxtFile:trCutAxis[0],TxtFile:pMoveC[0].trsf,TxtFile:tCfg)
            break

            case 2
              TxtFile:pLeave[0]=here(TxtFile:tCfg,TxtFile:fArray)
              if TxtFile:fPofffset.trsf=={0,0,0,0,0,0} and TxtFile:fToffset.trsf=={0,0,0,0,0,0}
                TxtFile:jLeave[0]=herej()
              else
                call Motion:Point2Joint(TxtFile:pLeave[0], TxtFile:jLeave[0],l_bRes)
                if !l_bRes
                  popUpMsg("Joint数据转换出错")
                endIf
              endIf
              call ExtAxis:RecordExtAxis(TxtFile:trLeaveAxis[0],TxtFile:pLeave[0].trsf,TxtFile:tCfg)

            break
          endSwitch


        endIf

      break







      //参数
      case 273
        //        l_bMoveL=TxtFile:bLeave[nLeaveIndex]
        //        call UI:Control_Para(TxtFile:trLeave,TxtFile:bLeave,false,TxtFile:nSingleType,nLeaveIndex,TxtFile:trLeaveAxis)
        //        //改变标志符
        //        if l_bMoveL!=TxtFile:bLeave[nLeaveIndex]
        //          //MOVEL
        //          if TxtFile:bLeave[nLeaveIndex]
        //            call Motion:Joint2Point(TxtFile:jLeave[nLeaveIndex],TxtFile:pLeave[nLeaveIndex])
        //          else
        //            //MOVEJ
        //            call Motion:Point2Joint(TxtFile:pLeave[nLeaveIndex], TxtFile:jLeave[nLeaveIndex],l_bRes)
        //            if !l_bRes
        //              popUpMsg("Joint数据转换出错")
        //            endIf
        //          endIf
        //
        //
        //          //2014.07.28记录同步外部轴
        //          if TxtFile:nSingleType==20
        //            call ExtAxis:RecordExtAxis(TxtFile:trLeaveAxis[0],TxtFile:pLeave[0].trsf,TxtFile:tCfg)
        //          endIf
        //
        //        endIf

        switch l_nIndex
          case 0
            call UI:Control_Para(TxtFile:trAppro,TxtFile:bAppro,false,TxtFile:nSingleType,0,TxtFile:trAppro)
          break

          case 1
            call UI:Control_Para(TxtFile:trCut,TxtFile:bMoveC,true,TxtFile:nSingleType,0,TxtFile:trCut)
          break
          case 2
            call UI:Control_Para(TxtFile:trLeave,TxtFile:bLeave,false,TxtFile:nSingleType,0,TxtFile:trLeaveAxis)
          break

        endSwitch
        TxtFile:bAppro[0]=TxtFile:bLeave[0]=TxtFile:bMoveC[0]=false


      break


      //      //删除
      //      case 274
      //        if size(TxtFile:pLeave)==1
      //          popUpMsg("离开点必须有一个")
      //        else
      //          call UI:Control_YesNO("确定要删除吗?",l_bRes)
      //          if l_bRes
      //            delete(TxtFile:pLeave[nLeaveIndex])
      //            delete(TxtFile:jLeave[nLeaveIndex])
      //            delete(TxtFile:bLeave[nLeaveIndex])
      //            delete(TxtFile:trLeave[nLeaveIndex])
      //            delete(TxtFile:trLeaveAxis[nLeaveIndex])
      //
      //          endIf
      //          TxtFile:trPointCount.z=size(TxtFile:pLeave)
      //          nLeaveIndex=min(TxtFile:trPointCount.z-1,nLeaveIndex)
      //
      //        endIf
      //
      //
      //      break


      //      模拟
      case 275
        call UI:Control_YesNO("确定要模拟吗?",l_bRes)
        if l_bRes
          DataBase:bKeyIO[0]= DataBase:bKeyIO[1]= DataBase:bKeyIO[2]=false
          //                    call TxtFile:RegulaPoint(true)
          //                    switch TxtFile:nSingleType
          //                      case 24
          //                        if TxtFile:trDownLead.rz<=0
          //                          call Algorith:GetArcAngle(TxtFile:pCut[0].trsf,TxtFile:pCut[1].trsf,TxtFile:pCut[2].trsf,TxtFile:trDownLead.rz,l_bRes)
          //                          TxtFile:trDownLead.rz=TxtFile:trDownLead.rz/10
          //                        endIf
          //                      break
          //                      case 12,2
          //                        if TxtFile:trDownLead.ry<=0
          //
          //                          TxtFile:trDownLead.ry=8
          //                        endIf
          //
          //                      break
          //                      case 10,20
          //                        if TxtFile:trPointCount.y<500
          //                          TxtFile:trPointCount.y=size(TxtFile:pCut)
          //                        endIf
          //
          //
          //                      break
          //
          //                    endSwitch

          // 个数赋值
          TxtFile:trPointCount.x=size(TxtFile:pAppro)
          TxtFile:trPointCount.z=size(TxtFile:pLeave)

          //                    //超过五百个点的情况
          //                    if (TxtFile:nSingleType!=10 and TxtFile:nSingleType!=20) or TxtFile:trPointCount.y<500
          //                      TxtFile:nReadCutCount=TxtFile:trPointCount.y
          call Simulate(-1)
          //                    else
          //先保存在模拟
          //  call Simulate(nTrajIndex+1)
          //                    endIf
          //   call TxtFile:RegulaPoint(false)
          call IO:SafteyIO()
          nPointType=3
          TxtFile:fArray.trsf={0,0,0,0,0,0}
          DataBase:bKeyIO[0]= DataBase:bKeyIO[1]= DataBase:bKeyIO[2]=false
          call UI:Control_PanelMd("模拟结束")
          delay(2)
        endIf

        cls()
      break




      //保存
      case 278
        //        //计算总个数
        //        TxtFile:trPointCount.y=0
        //        for l_nNum=0 to size(TxtFile:nPartTrajCount)-1
        //          TxtFile:trPointCount.y=TxtFile:trPointCount.y+TxtFile:nPartTrajCount[l_nNum]
        //        endFor
        //        if TxtFile:trPointCount.y==0
        //          TxtFile:trPointCount.y=size(TxtFile:pCut)
        //        endIf

        //保存
        DataBase:bStopPoll=true
        TxtFile:trPointCount.y=TxtFile:trPointCount.x=TxtFile:trPointCount.z=1
        call UI:Control_YesNO("确定要保存吗?",l_bRes)
        if l_bRes
          call UI:Control_PanelMd("请等待，正在保存...")
          call TxtFile:SaveTraj(l_bRes)
          if !l_bRes
            popUpMsg("保存路径文件出错")
          else
            call TxtFile:EditRecipe(TxtFile:nTrajIndex,false,l_bRes)
            if !l_bRes
              popUpMsg("保存生产文件出错")
            else
              call TxtFile:ReadProduct("Disk://Txt/Recipe.txt",TxtFile:sProductName,true,l_bRes)
              if !l_bRes
                popUpMsg("读取生产文件出错")
              else
                popUpMsg("保存成功")
                bSaveTxt=true
              endIf
            endIf
          endIf
        endIf
        call TxtFile:CloseFile()
        cls()


      break



      //      //返回
      //      case 277
      //        nPointType=2
      //      break

      //退出
      case 276
        if bSaveTxt
          call UI:Control_YesNO("确定要退出吗?",l_bRes)
        else
          call UI:Control_YesNO("路径没有被保存,确定要退出吗?",l_bRes)
        endIf
        if l_bRes
          nPointType=-1
          return
        endIf
      break

      //点位
      case 270
        //        if TxtFile:bLeave[nLeaveIndex]
        //          call UI:Control_Point(TxtFile:pLeave[nLeaveIndex] )
        //        else
        //          call UI:Control_Joint(TxtFile:jLeave[nLeaveIndex])
        //        endIf

        switch l_nIndex
          case 0
            call UI:Control_Joint(TxtFile:jAppro[0])
          break

          case 1
            call UI:Control_Point(TxtFile:pCut[0])
          break


          case 2
            call UI:Control_Joint(TxtFile:jLeave[0])
          break


        endSwitch

        cls()
      break

    endSwitch
    if (l_nKey<279 and l_nKey>=260)or l_nKey==112 or !l_bFirst
      nApproIndex=nCutIndex=nLeaveIndex=0
      call SingleMove(l_nIndex+1)
      l_bFirst=true
      //      call GetListItems()
      resize(sSItem,1,3)
      sSItem[0]="1.MOVEJ"
      sSItem[1]="2.MOVEL"
      sSItem[2]="3.MOVEJ"
      call UI:Form_PanelList("LasMAN3.6->示教路径","空走路径点",sSItem,l_nIndex,",记录,参数,,模拟,退出,,保存")
      call UI:Control_Mess("类型:"+TxtFile:sTrajType[TxtFile:nSingleType],"")





    endIf


    //2014.07.30
    //同步七八轴
    if (TxtFile:bSync7Axis or TxtFile:bSync8Axis)
      call ExtAxis:RecordExtAxis(l_trTrsf,l_trTrsf,TxtFile:tCfg)

      gotoxy(1,12)
      put("七轴:"+toString(".3",l_trTrsf.x))
      if TxtFile:bSync8Axis
        gotoxy(20,12)
        put("八轴:"+toString(".3",l_trTrsf.y))
      endIf
    endIf
    //



    delay(0)
    DataBase:bStopPoll=false
  endWhile



end

--- IsPointOK.pgx ---
public program IsPointOK(num x_nIndex, num x_nType, num x_nMC, bool& x_bRes)
  local num l_nNum
  local pointRx l_pPBuff
  local pointRx l_pHere
  local jointRx l_jJ
begin

  //判断点位是否可以走到
  //主要是MOVEC和MOVEL点


  //2014.12.05
  if (TxtFile:nSingleType==20 or TxtFile:nSingleType==9) and ExtAxis:bMoveType
    x_bRes=true
    return
  endIf


  x_bRes=false
  l_pHere=here(TxtFile:tCfg,TxtFile:fArray)

  switch x_nType

    //趋近
    case 1
      for l_nNum=0.1 to 1 step 0.1
        link(l_pPBuff,world)
        l_pPBuff.trsf={0,0,0,0,0,0}
        l_pPBuff.trsf=interpolateL(l_pHere.trsf,TxtFile:pAppro[x_nIndex].trsf,l_nNum)
        link(l_pPBuff,TxtFile:fArray)
        x_bRes=pointToJoint(TxtFile:tCfg,herej(),l_pPBuff,l_jJ)
        if !x_bRes
          return
        endIf
        x_bRes=isInRange(l_jJ)
        if !x_bRes
          return
        endIf
      endFor
    break

    //切割
    case 2
      if !TxtFile:bMoveC[x_nIndex] or (x_nMC!=0 and TxtFile:bMoveC[x_nIndex])



        for l_nNum=0.1 to 1 step 0.1
          link(l_pPBuff,world)
          l_pPBuff.trsf={0,0,0,0,0,0}
          if !TxtFile:bMoveC[x_nIndex] or (x_nMC==2 and TxtFile:bMoveC[x_nIndex])
            l_pPBuff.trsf=interpolateL(l_pHere.trsf,TxtFile:pCut[x_nIndex].trsf,l_nNum)
          else
            //圆弧中间点
            l_pPBuff.trsf=interpolateL(l_pHere.trsf,TxtFile:pMoveC[x_nIndex].trsf,l_nNum)

          endIf
          link(l_pPBuff,TxtFile:fArray)
          x_bRes=pointToJoint(TxtFile:tCfg,herej(),l_pPBuff,l_jJ)
          if !x_bRes
            return
          endIf
          x_bRes=isInRange(l_jJ)
          if !x_bRes
            return
          endIf
        endFor
      else

        //2014.11.28
        //对于x_nIndex=0,则直接跳出
        if x_nIndex<1
          x_bRes=true
          return
        endIf



        //中间点一定必须是钝角
        l_pHere=TxtFile:pCut[x_nIndex-1]
        if TxtFile:pMoveC[x_nIndex].trsf==TxtFile:pCut[x_nIndex].trsf or l_pHere.trsf==TxtFile:pCut[x_nIndex].trsf or l_pHere.trsf==TxtFile:pMoveC[x_nIndex].trsf
          x_bRes=false
          return
        endIf
        l_nNum=power(distance(l_pHere.trsf,TxtFile:pMoveC[x_nIndex].trsf),2)+power(distance(TxtFile:pCut[x_nIndex].trsf,TxtFile:pMoveC[x_nIndex].trsf),2)
        if l_nNum>power(distance(l_pHere.trsf,TxtFile:pCut[x_nIndex].trsf),2)
          x_bRes=false
          return
        endIf

        for l_nNum=0.1 to 1 step 0.1
          link(l_pPBuff,world)
          l_pPBuff.trsf={0,0,0,0,0,0}
          if  nCutIndex>nCursonIndex
            l_pPBuff.trsf=interpolateC(TxtFile:pCut[x_nIndex].trsf,TxtFile:pMoveC[x_nIndex].trsf,l_pHere.trsf,l_nNum)
          else
            l_pPBuff.trsf=interpolateC(l_pHere.trsf,TxtFile:pMoveC[x_nIndex].trsf,TxtFile:pCut[x_nIndex].trsf,l_nNum)

          endIf

          link(l_pPBuff,TxtFile:fArray)
          x_bRes=pointToJoint(TxtFile:tCfg,herej(),l_pPBuff,l_jJ)
          if !x_bRes
            return
          endIf
          x_bRes=isInRange(l_jJ)
          if !x_bRes
            return
          endIf
        endFor

      endIf






    break
    //离开
    case 3
      for l_nNum=0.1 to 1 step 0.1
        link(l_pPBuff,world)
        l_pPBuff.trsf={0,0,0,0,0,0}
        l_pPBuff.trsf=interpolateL(l_pHere.trsf,TxtFile:pLeave[x_nIndex].trsf,l_nNum)
        link(l_pPBuff,TxtFile:fArray)
        x_bRes=pointToJoint(TxtFile:tCfg,herej(),l_pPBuff,l_jJ)
        if !x_bRes
          return
        endIf
        x_bRes=isInRange(l_jJ)
        if !x_bRes
          return
        endIf
      endFor
    break
  endSwitch
  x_bRes=true



end

--- LEAVE.pgx ---
public program Leave()
  local num l_nKey
  local bool l_bRes
  local string l_sProductName
  local jointRx l_jJBuff
  local bool l_bCut
  local bool l_bMoveL
  local num l_nNum
  local num l_nApproCount
  local bool l_bFirst
  local trsf l_trTrsf
  local num l_nToolMode
  local num l_nAtPosition
begin
  //离开点界面
  DataBase:bMoveTask=false
  call IO:KeyDigtalIO(false,false,false,0,0)
  TxtFile:nWeldActionId=0
  TxtFile:fArray.trsf={0,0,0,0,0,0}
  //2014.2.17  在哪个坐标系中运动
  if !DataBase:bWorldMove
    $jogContext(TxtFile:tCfg,TxtFile:fArray,0)
  else
    $jogContext(TxtFile:tCfg,world,0)
  endIf


  //第一次示教,是否需要回退点
  if bFirstTeach==false
    bFirstTeach=true
    if TxtFile:bMoveBack
      l_nApproCount=size(TxtFile:pAppro)
      resize(TxtFile:pLeave,1,l_nApproCount)
      resize(TxtFile:jLeave,1,l_nApproCount)
      resize(TxtFile:bLeave,1,l_nApproCount)
      resize(TxtFile:trLeave,1,l_nApproCount)
      resize(TxtFile:trLeaveAxis,1,l_nApproCount)

      for l_nNum=0 to l_nApproCount-1
        TxtFile:bLeave[l_nNum]=TxtFile:bAppro[l_nApproCount-1-l_nNum]
        TxtFile:jLeave[l_nNum]=TxtFile:jAppro[l_nApproCount-1-l_nNum]
        TxtFile:pLeave[l_nNum]=TxtFile:pAppro[l_nApproCount-1-l_nNum]
        TxtFile:trLeave[l_nNum]=TxtFile:trAppro[l_nApproCount-1-l_nNum]

        TxtFile:trLeaveAxis[l_nNum]=TxtFile:trApproAxis[l_nApproCount-1-l_nNum]

      endFor

    endIf

  endIf

  TxtFile:trPointCount.z=size(TxtFile:pLeave)

  //界面初始化
  nPointType=3
  cls()
  while  nPointType==3
    l_nKey=getKey()
    DataBase:bMoveTask=false
    TxtFile:nWeldActionId=0
    switch l_nKey

      //配置
      case 112
        call SetTrajPara()

      break



      case 261
        nLeaveIndex=max(nLeaveIndex-1,0)


      break


      case 266
        nLeaveIndex=min(nLeaveIndex+1,size(TxtFile:pLeave)-1)


      break
      //向左
      case 264
        //2015.08.16

        nPointType=2

      break

      //插入
      case 271

        insert(TxtFile:pLeave[nLeaveIndex+1])
        insert(TxtFile:jLeave[nLeaveIndex+1])
        insert(TxtFile:bLeave[nLeaveIndex+1])
        insert(TxtFile:trLeave[nLeaveIndex+1])
        insert(TxtFile:trLeaveAxis[nLeaveIndex+1])

        TxtFile:pLeave[nLeaveIndex+1]=TxtFile:pLeave[nLeaveIndex]
        TxtFile:jLeave[nLeaveIndex+1]=TxtFile:jLeave[nLeaveIndex]
        TxtFile:bLeave[nLeaveIndex+1]=TxtFile:bLeave[nLeaveIndex]
        TxtFile:trLeave[nLeaveIndex+1]=TxtFile:trLeave[nLeaveIndex]
        TxtFile:trLeaveAxis[nLeaveIndex+1]=TxtFile:trLeaveAxis[nLeaveIndex]
        nLeaveIndex=nLeaveIndex+1

        TxtFile:trPointCount.z=size(TxtFile:pLeave)
        //2014.05.30
        //××××××××××××××××××××××××××××××××××××××8
        if TxtFile:nSingleType!=20 and TxtFile:nSingleType!=9
          TxtFile:pLeave[nLeaveIndex]=here(TxtFile:tCfg,TxtFile:fArray)
          if TxtFile:fPofffset.trsf=={0,0,0,0,0,0} and TxtFile:fToffset.trsf=={0,0,0,0,0,0}
            TxtFile:jLeave[nLeaveIndex]=herej()
          else
            call Motion:Point2Joint(TxtFile:pLeave[nLeaveIndex], TxtFile:jLeave[nLeaveIndex],l_bRes)
            if !l_bRes
              popUpMsg("Joint数据转换出错")
            endIf
          endIf
        endIf

        //×××××××××××××××××××××××××××××××××××××××××





      break


      //记录
      case 272
        TxtFile:fArray.trsf={0,0,0,0,0,0}
        //2015.08.10
        l_bRes=true
        // call UI:Control_YesNO("确定要记录吗?",l_bRes)
        if l_bRes
          TxtFile:pLeave[nLeaveIndex]=here(TxtFile:tCfg,TxtFile:fArray)
          if TxtFile:fPofffset.trsf=={0,0,0,0,0,0} and TxtFile:fToffset.trsf=={0,0,0,0,0,0}
            TxtFile:jLeave[nLeaveIndex]=herej()
          else
            call Motion:Point2Joint(TxtFile:pLeave[nLeaveIndex], TxtFile:jLeave[nLeaveIndex],l_bRes)
            if !l_bRes
              popUpMsg("Joint数据转换出错")
            endIf
          endIf
          //2014.07.28记录同步外部轴
          if TxtFile:nSingleType==20 or TxtFile:nSingleType==9
            call ExtAxis:RecordExtAxis(TxtFile:trLeaveAxis[nLeaveIndex],TxtFile:pLeave[nLeaveIndex].trsf,TxtFile:tCfg)
          endIf

        endIf

      break

      //参数
      case 273
        l_bMoveL=TxtFile:bLeave[nLeaveIndex]
        call UI:Control_Para(TxtFile:trLeave,TxtFile:bLeave,false,TxtFile:nSingleType,nLeaveIndex,TxtFile:trLeaveAxis)
        //改变标志符
        if l_bMoveL!=TxtFile:bLeave[nLeaveIndex]
          //MOVEL
          if TxtFile:bLeave[nLeaveIndex]
            call Motion:Joint2Point(TxtFile:jLeave[nLeaveIndex],TxtFile:pLeave[nLeaveIndex])
          else
            //MOVEJ
            call Motion:Point2Joint(TxtFile:pLeave[nLeaveIndex], TxtFile:jLeave[nLeaveIndex],l_bRes)
            if !l_bRes
              popUpMsg("Joint数据转换出错")
            endIf
          endIf


          //2014.07.28记录同步外部轴
          if TxtFile:nSingleType==20 or TxtFile:nSingleType==9
            call ExtAxis:RecordExtAxis(TxtFile:trLeaveAxis[nLeaveIndex],TxtFile:pLeave[nLeaveIndex].trsf,TxtFile:tCfg)
          endIf

        endIf
      break

      //删除
      case 274
        if size(TxtFile:pLeave)==1
          popUpMsg("离开点必须有一个")
        else
          call UI:Control_YesNO("确定要删除吗?",l_bRes)
          if l_bRes
            delete(TxtFile:pLeave[nLeaveIndex])
            delete(TxtFile:jLeave[nLeaveIndex])
            delete(TxtFile:bLeave[nLeaveIndex])
            delete(TxtFile:trLeave[nLeaveIndex])
            delete(TxtFile:trLeaveAxis[nLeaveIndex])

          endIf
          TxtFile:trPointCount.z=size(TxtFile:pLeave)
          nLeaveIndex=min(TxtFile:trPointCount.z-1,nLeaveIndex)

        endIf


      break
      //模拟
      case 275
        call UI:Control_YesNO("确定要模拟吗?",l_bRes)
        if l_bRes
          DataBase:bKeyIO[0]= DataBase:bKeyIO[1]= DataBase:bKeyIO[2]=false
          call TxtFile:RegulaPoint(true)
          switch TxtFile:nSingleType
            case 24
              if TxtFile:trDownLead.rz<=0
                call Algorith:GetArcAngle(TxtFile:pCut[0].trsf,TxtFile:pCut[1].trsf,TxtFile:pCut[2].trsf,TxtFile:trDownLead.rz,l_bRes)
                TxtFile:trDownLead.rz=TxtFile:trDownLead.rz/10
              endIf
            break
            case 12,2
              if TxtFile:trDownLead.ry<=0

                TxtFile:trDownLead.ry=8
              endIf

            break
            case 10,20
              if TxtFile:trPointCount.y<500
                TxtFile:trPointCount.y=size(TxtFile:pCut)
              endIf


            break

          endSwitch

          //个数赋值
          TxtFile:trPointCount.x=size(TxtFile:pAppro)
          TxtFile:trPointCount.z=size(TxtFile:pLeave)

          //超过五百个点的情况
          if (TxtFile:nSingleType!=10 and TxtFile:nSingleType!=20) or TxtFile:trPointCount.y<500
            TxtFile:nReadCutCount=TxtFile:trPointCount.y
            call Simulate(-1)
          else
            //先保存在模拟
            call Simulate(nTrajIndex+1)
          endIf
          call TxtFile:RegulaPoint(false)
          call IO:SafteyIO()
          nPointType=3
          TxtFile:fArray.trsf={0,0,0,0,0,0}
          DataBase:bKeyIO[0]= DataBase:bKeyIO[1]= DataBase:bKeyIO[2]=false
          call UI:Control_PanelMd("模拟结束")
          delay(2)

        endIf

        //        //*************************
        //        //20150616
        //        //如果不是远程模式，则等待按下
        //        //安全机制
        //        DataBase:nToolMode=workingMode()
        //        l_nToolMode=-1
        //        if DataBase:nToolMode!=4
        //          while l_nToolMode!=6
        //            DataBase:nToolMode=workingMode(l_nToolMode)
        //            delay(0)
        //          endWhile
        //        endIf
        //        //**************************

        //2015.12.30
        //安全因素进行切换
        while workingMode()!=1
          popUpMsg("请先切换到手动模式,然后点击OK")
          delay(0.1)
        endWhile



        cls()
      break




      //保存
      case 278
        //计算总个数
        TxtFile:trPointCount.y=0
        for l_nNum=0 to size(TxtFile:nPartTrajCount)-1
          TxtFile:trPointCount.y=TxtFile:trPointCount.y+TxtFile:nPartTrajCount[l_nNum]
        endFor
        if TxtFile:trPointCount.y==0
          TxtFile:trPointCount.y=size(TxtFile:pCut)
        endIf

        //保存
        DataBase:bStopPoll=true
        call UI:Control_YesNO("确定要保存吗?",l_bRes)
        if l_bRes
          call UI:Control_PanelMd("请等待，正在保存...")
          call TxtFile:SaveTraj(l_bRes)
          if !l_bRes
            popUpMsg("保存路径文件出错")
          else
            call TxtFile:EditRecipe(TxtFile:nTrajIndex,false,l_bRes)
            if !l_bRes
              popUpMsg("保存生产文件出错")
            else
              call TxtFile:ReadProduct("Disk://Txt/Recipe.txt",TxtFile:sProductName,true,l_bRes)
              if !l_bRes
                popUpMsg("读取生产文件出错")
              else
                popUpMsg("保存成功")
                bSaveTxt=true
              endIf
            endIf
          endIf
        endIf
        call TxtFile:CloseFile()
        cls()


      break



      //返回
      case 277
        nPointType=2
      break

      //退出
      case 276
        if bSaveTxt
          call UI:Control_YesNO("确定要退出吗?",l_bRes)
        else
          call UI:Control_YesNO("路径没有被保存,确定要退出吗?",l_bRes)
        endIf
        if l_bRes
          nPointType=-1
          return
        endIf
      break

      //点位
      case 270
        if TxtFile:bLeave[nLeaveIndex]
          call UI:Control_Point(TxtFile:pLeave[nLeaveIndex] )
        else
          call UI:Control_Joint(TxtFile:jLeave[nLeaveIndex])
        endIf
        cls()
      break

    endSwitch
    if (l_nKey<279 and l_nKey>=260)or l_nKey==112 or !l_bFirst
      call SingleMove(3)
      l_bFirst=true
      call GetListItems()
      call UI:Form_PanelList("LasMAN3.6->示教路径","离开点",sSItem,nLeaveIndex,"插入,记录,参数,删除,模拟,退出,返回,保存")
      call UI:Control_Mess("类型:"+TxtFile:sTrajType[TxtFile:nSingleType],"离开点个数:"+toString("",size(TxtFile:pLeave)))





    endIf

    //2014.07.30
    //同步七八轴
    if TxtFile:nSingleType==20 and (TxtFile:bSync7Axis or TxtFile:bSync8Axis)
      call ExtAxis:RecordExtAxis(l_trTrsf,l_trTrsf,TxtFile:tCfg)

      gotoxy(1,12)
      put("七轴:"+toString(".3",l_trTrsf.x))
      if TxtFile:bSync8Axis
        gotoxy(20,12)
        put("八轴:"+toString(".3",l_trTrsf.y))
      endIf
    endIf
    //


    //为了表示到达位置
    //2015.08.10
    //为整个列表进行修改

    if nLeaveIndex>10
      l_nAtPosition=nLeaveIndex-10
    else
      l_nAtPosition=0
    endIf

    for l_nNum=0 to min(size(TxtFile:bLeave)-1,10)
      gotoxy(22,min(l_nNum+1,10))

      //  setTextMode(1)
      setTextMode(sel((l_nAtPosition+l_nNum)==nLeaveIndex,1,0))
      if TxtFile:bLeave[nLeaveIndex]
        if distance(TxtFile:pLeave[l_nAtPosition+l_nNum],here(TxtFile:tFileTool,TxtFile:fArray))<0.1
          put("@")
        else
          put("│")
        endIf

      else
        if distance(jointToPoint(TxtFile:tFileTool,TxtFile:fArray,herej()),jointToPoint(TxtFile:tFileTool,TxtFile:fArray,TxtFile:jLeave[l_nAtPosition+l_nNum]))<0.1
          put("@")
        else
          put("│")
        endIf
      endIf
    endFor


    //*************************





    delay(0)
    DataBase:bStopPoll=false
  endWhile



end

--- ONACTION.pgx ---
program OnAction()
  local num l_nX
  local num l_nY
begin
  //示教动作
  //示教动作执行

  wait(isPowered())
  for l_nX=0 to 11
    for l_nY=0 to 1
     Motion:nMoveidAction[l_nX,l_nY]=TxtFile:nAction[nTeachAction,l_nX,l_nY]

    endFor
  endFor


  call IO:Action(Motion:nMoveidAction,true,-1)
  call IO:Action(Motion:nMoveidAction,false,-1)


end

--- OneWpMproChoose.pgx ---
public program OneWpMproChoose()
  local num l_nNum
  local num l_nProductIndex
  local string l_sSFileName
  local bool l_bRes
begin
  //同工位多产品选择
  //TxtFile:bMoreProd1Wp

  //bMultiNormal  多产品合并为一个工位


  //参数初始化
  for l_nNum=0 to size(DataBase:sProductName)-1
    DataBase:sProductName[l_nNum]=""
  endFor

  //选择产品
  //    for l_nNum=1 to DataBase:nWorkPlaceCount
  //
  l_nNum=DataBase:nWorkPlaceIndex
  if !DataBase:bMultiNormal
    //为法利莱
    call IO:ChooseMultPro(l_nNum,l_nProductIndex)
  else
    //为大族
    call IO:ChoosehansPro(l_nNum,DataBase:nProductIndex,DataBase:nWpMutiCount)
    l_nProductIndex=DataBase:nProductIndex
  endIf




  //选择不正确则退出
  l_sSFileName="Disk://Txt/"+toString("",l_nNum)+"Product"+toString("",l_nProductIndex)+".txt"
  if l_nProductIndex<1
    DataBase:nInterfaceType=9
    return
  endIf

  if  $fileExists(l_sSFileName)==false
    DataBase:nInterfaceType=9
    popUpMsg(l_sSFileName+"文件不存在")
    logMsg(l_sSFileName+"文件不存在")
    return
  endIf

  //读取文件名
  DataBase:bStopPoll=true
  call TxtFile:ReadProductName(l_sSFileName,l_bRes)
  DataBase:bStopPoll=false
  if l_bRes
    DataBase:sProductName[l_nNum]=TxtFile:sProductName
  else
    DataBase:nInterfaceType=9
    popUpMsg("读取产品名出错")
    logMsg(l_sSFileName+"产品名出错")
    disablePower()
    return
  endIf

  //拷贝
  call TxtFile:CloseFile()
  if $fileExists("Disk://Txt/Product"+toString("",l_nNum)+".txt")
    $delete("Disk://Txt/Product"+toString("",l_nNum)+".txt")
  endIf
  if !$copy(l_sSFileName,"Disk://Txt/Product"+toString("",l_nNum)+".txt")
    DataBase:nInterfaceType=9
    popUpMsg("拷贝文件出错")
    logMsg("拷贝产品名出错")
    return
  endIf
  //
  //    endFor
  //

  //把工位值赋给
  DataBase:nWorkPlaceIndex=l_nNum


end

--- PRODUCT.pgx ---
program Product()
  local num l_nNum
  local bool l_bRes
  local num l_nTime
  local joint l_jJ
  local num l_nKey
begin
  //生产函数


  //变量初始化
  DataBase:nWorkPlaceIndex=0
  DataBase:nCycleIndex=0
  bPowerFlag=false
  DataBase:nCycleCount=max(1,DataBase:nCycleCount)


  //等待机械手臂上电
  if !isPowered()
    call GetProductMess("等待上电")
    wait(DataBase:bPowerOn and isPowered())
  endIf

  bPowerFlag=true



  //标志符响应

  while DataBase:nInterfaceType==13

    //检查机械手臂是否在零位
    // l_jJ=herej()
    //l_nKey= abs(l_jJ.j1-TxtFile:jHome.j1)+abs(l_jJ.j2-TxtFile:jHome.j2)+abs(l_jJ.j3-TxtFile:jHome.j3)
    // l_nKey=l_nKey+ abs(l_jJ.j4-TxtFile:jHome.j4)+abs(l_jJ.j5-TxtFile:jHome.j5)+abs(l_jJ.j6-TxtFile:jHome.j6)


    //    if l_nKey>0.3
    //      popUpMsg("机械手臂请回到零位")
    //      return
    //    endIf

    if distance(here(TxtFile:tCfg,world),jointToPoint(TxtFile:tCfg,world,TxtFile:jHome))>1
      popUpMsg("机械手臂请回到零位")
      return
    endIf


    //机械手臂在安全点位置
    call IO:AtHome(true)

    //等待按钮触发

    TxtFile:nReadTrajIndex=0


    //产品与工位选择
    call WorkPlaceChose()


    //机械手臂在安全点位置
    call IO:AtHome(false)


    //报错机制,
    if DataBase:nWorkPlaceIndex<1 or DataBase:nWorkPlaceIndex>DataBase:nWorkPlaceCount
      DataBase:nInterfaceType=9
      logMsg("生产结束")
      return
    endIf


    //如果多于一个工位或者同工位多产品，则读取文件
    DataBase:bStopPoll=true
    if DataBase:nWorkPlaceCount>1 or TxtFile:bMoreProd1Wp
      //读取路径名

      call TxtFile:ReadProduct("Disk://Txt/Product"+toString("",DataBase:nWorkPlaceIndex)+".txt",DataBase:sProductName[DataBase:nWorkPlaceIndex],false,l_bRes)

      //路径个数必须大于或者等于1
      if !l_bRes or TxtFile:nTotalTraj<1
        popUpMsg("读取工位"+toString("",DataBase:nWorkPlaceIndex)+"生产文件出错")
        return
      endIf
    endIf

    //如果读取文件中的PresetName
    if TxtFile:sPresetName!="StaubliPreset"
      call TxtFile:ReadMatchPreset("Disk://Txt/Preset"+toString("",DataBase:nWorkPlaceIndex)+".txt",TxtFile:sPresetName,l_bRes)
    endIf


    //开始生产
    DataBase:bStopPoll=false
    call IO:Light(2)
    call GetProductMess("工位"+toString("",DataBase:nWorkPlaceIndex)+"开始启动")
    call GetProductMess("开始生产"+DataBase:sProductName[DataBase:nWorkPlaceIndex])
    logMsg("工位"+toString("",DataBase:nWorkPlaceIndex)+"生产"+DataBase:sProductName[DataBase:nWorkPlaceIndex])



    //2014.4.16
    //每个工位的值加,计数
    //用户上位机进行统计使用

    DataBase:nWpProduct[DataBase:nWorkPlaceIndex]=DataBase:nWpProduct[DataBase:nWorkPlaceIndex]+1
    DataBase:nProductCount=DataBase:nProductCount+1


    //路径过滤
    if TxtFile:bTrajFilter
      call GetProductMess("信号控制路径过滤")
    endIf

    //产品生产前的动作
    call Custom:BeforeProduct(DataBase:nWorkPlaceIndex)


    //生产的总个数
    Motion:nStartTraj=1
    Motion:nEndTraj=TxtFile:nTotalTraj
    l_nTime=clock()




    //建立两个任务
    if taskStatus("ReadFile")!=-1
      taskKill("ReadFile")
    endIf

    if taskStatus("Preset")!=-1
      taskKill("Preset")
    endIf


    if taskStatus("WeldEnd")!=-1
      taskKill("WeldEnd")
    endIf
    TxtFile:bReadProduct=true
    taskCreate "ReadFile",100,Motion:ReadTraj()
    delay(0)
    taskCreate "Preset",100,Motion:Preset()


    if TxtFile:bWeldEnable
      taskCreateSync "WeldEnd",0.004,bSyc,Motion:WeldEnd()
    endIf

    delay(0)



    //机器人运动
    call Motion:Move()

    //结束生产
    TxtFile:bReadProduct=false
    if taskStatus("ReadFile")!=-1
      taskKill("ReadFile")
    endIf

    if taskStatus("Preset")!=-1
      taskKill("Preset")
    endIf

    if taskStatus("WeldEnd")!=-1
      taskKill("WeldEnd")
    endIf


    //工位完成,发出信号
    waitEndMove()
    //l_jJ=herej()
    // l_nNum=abs(l_jJ.j1-TxtFile:jHome.j1)+abs(l_jJ.j2-TxtFile:jHome.j2)+abs(l_jJ.j3-TxtFile:jHome.j3)
    // l_nNum=l_nNum+abs(l_jJ.j4-TxtFile:jHome.j4)+abs(l_jJ.j5-TxtFile:jHome.j5)+abs(l_jJ.j6-TxtFile:jHome.j6)


    //生产中途退出
    //if l_nNum>0.3
    //  return
    // endIf

    //2014.12.08
    //代码重构
    //如果与安全点距离大于1mm,则跳出循环
    if distance(here(TxtFile:tCfg,world),jointToPoint(TxtFile:tCfg,world,TxtFile:jHome))>1
      return
    endIf


    //输出工位完成信息
    //**************************
    //2015.04.20
    call IO:WorkPlaceFinish(0)





    //多工位多产品
    if (DataBase:bMultiNormal and TxtFile:bMoreProd1Wp and DataBase:nWorkPlaceIndex>=DataBase:nWpProduct[DataBase:nWorkPlaceIndex]) and DataBase:bWpFinishIOOut
      call IO:WorkPlaceFinish(DataBase:nWorkPlaceIndex)
    endIf


    //一般情况下的
    //多工位多产品
    if !TxtFile:bMoreProd1Wp and !DataBase:bExtraContrAxis  and DataBase:bWpFinishIOOut
      call IO:WorkPlaceFinish(DataBase:nWorkPlaceIndex)
    endIf

    //外部PLC控制第七轴运动，到底home位置时发出工位完成信号
    if DataBase:bExtraContrAxis
      call IO:AtHomePulse()
    endIf


    //**************************************

    //生产IO初始化
    call IO:WaitProIOEnd(DataBase:nWorkPlaceIndex)
    //DataBase:bCanProduct[DataBase:nWorkPlaceIndex]=false
    //生产结束
    call GetProductMess("结束生产"+DataBase:sProductName[DataBase:nWorkPlaceIndex-1])
    DataBase:nCycleTime=clock()-l_nTime

    //生产完成之后
    call Custom:AfterWorkPlace(DataBase:nWorkPlaceIndex)

  endWhile


end

--- SetTrajPara.pgx ---
program SetTrajPara()
  local bool l_bCut
  local num l_nNum
  local trsf l_trTrsf
  local trsf l_trTSource[3]
  local bool l_bRes
  local num l_nDia
  local num l_nLength[2]
begin

  //设置路径参数
  //主要是在appro,cut,leave界面中的 p按钮使用
  //参数预设



  //三点规则图形
  if TxtFile:nSingleType!=12 and TxtFile:nSingleType!=10 and  TxtFile:nSingleType!=2 and TxtFile:nSingleType!=20

    //算圆弧度
    if TxtFile:trDownLead.rz<=0 and TxtFile:nSingleType==24
      call Algorith:GetArcAngle(TxtFile:pCut[0].trsf,TxtFile:pCut[1].trsf,TxtFile:pCut[2].trsf,l_nNum,l_bRes)
      TxtFile:trDownLead.rz=l_nNum/10
    endIf


    //算直径
    l_trTSource[0]=TxtFile:pCut[0].trsf
    l_trTSource[1]=TxtFile:pCut[1].trsf
    l_trTSource[2]=TxtFile:pCut[2].trsf

    call Algorith:Circumcircle(l_trTSource,l_trTrsf,l_nDia,l_bRes)
    if l_bRes
      TxtFile:trDownLead.ry=l_nDia
    endIf

    //算边长
    l_nLength[0]=distance(l_trTSource[0],l_trTSource[1])
    l_nLength[1]=distance(l_trTSource[2],l_trTSource[1])


  else
    if TxtFile:trDownLead.ry<=0
      TxtFile:trDownLead.ry=8
    endIf


  endIf




  //设置内切与外切
  //图形类型小于10的才有内切外切之说
  l_bCut=TxtFile:nSingleType<10

  if TxtFile:bWeldEnable
    //焊接中不用到异步八轴
    l_bCut=TxtFile:trWorkplace.z==1
  endIf


  //参数设置
  call UI:Control_Traj(TxtFile:fTraj.trsf,TxtFile:fToffset.trsf,TxtFile:trArray,TxtFile:trDownLead,TxtFile:trWorkplace,l_bCut,TxtFile:nTrajDelay,l_nLength,TxtFile:bWeldEnable)


  if TxtFile:nSingleType!=10 and l_bCut!=(TxtFile:nSingleType<10) and TxtFile:nSingleType!=20
      TxtFile:nSingleType=TxtFile:nSingleType+sel(l_bCut,-10,10)
  endIf

    if TxtFile:bWeldEnable
      TxtFile:trWorkplace.z=sel( l_bCut,1,0)
    endIf



  //修改路径点的位置
  //三点法根据直径修改位置

  if TxtFile:nSingleType!=12 and TxtFile:nSingleType!=10 and  TxtFile:nSingleType!=2 and TxtFile:nSingleType!=20
    call Algorith:ChangeLength(TxtFile:pCut,l_nLength)

    TxtFile:trDownLead.ry=max(0.001,TxtFile:trDownLead.ry)
    if l_nDia!=TxtFile:trDownLead.ry
      l_trTSource[0]=TxtFile:pCut[0].trsf
      l_trTSource[1]=TxtFile:pCut[1].trsf
      l_trTSource[2]=TxtFile:pCut[2].trsf

      call Algorith:Circumcircle(l_trTSource,l_trTrsf,l_nDia,l_bRes)
      if !l_bRes
        return
      endIf

      for l_nNum=0 to 2
        call Algorith:ChangeCirPoint(l_trTrsf,TxtFile:trDownLead.ry,TxtFile:pCut[l_nNum].trsf,TxtFile:pCut[sel(l_nNum==2,0,l_nNum+1)].trsf,l_bRes)
        if !l_bRes
          return
        endIf

      endFor
    endIf





  endIf

end

--- SIMULATE.pgx ---
public program Simulate(num x_nTrajIndex)
  local num l_nKey
  local num l_nPointType
  local num l_nPointIndex
  local bool l_bRes
  local string l_sItemTitle
  local bool l_bKeyIO[3]
  local num l_nNum
  local num l_nID
  local num l_nToolMode
  local trsf l_trArray
begin

  logMsg(TxtFile:sProductName+"开始模拟"+toString("",x_nTrajIndex))
  if x_nTrajIndex>=0
    call UI:Control_PanelMd("请等待，正在读取文件......")
  else
    call UI:Control_PanelMd("请等待，开始模拟......")
  endIf



  //参数初始化
  DataBase:bIOStart=false


  // DataBase:bKeyIO[0]= DataBase:bKeyIO[1]= DataBase:bKeyIO[2]=false
  DataBase:nPointType=0
  DataBase:nID=0
  nPointType=-1
  l_nPointIndex=0
  nApproIndex=0
  nCutIndex=0
  nLeaveIndex=0
  n500Count=0

  setMoveId(0)

  //2015.12.30
  //需要建立task之前，先kill
  taskKill("Simulation")
  wait(taskStatus("Simulation")==-1)



  //建立路径
  if x_nTrajIndex==-1
    taskCreate "Simulation",100,Motion:TeachSimu(0,0)
  else
    if x_nTrajIndex==-2
      taskCreate "Simulation",100,Motion:TeachSimu(DataBase:nPartMove[0],DataBase:nPartMove[1])
    else
      taskCreate "Simulation",100,Motion:TrajSimu(x_nTrajIndex)
    endIf
  endIf
  l_bKeyIO[0]=DataBase:bKeyIO[0]
  l_bKeyIO[1]=DataBase:bKeyIO[1]
  l_bKeyIO[2]=DataBase:bKeyIO[2]

  delay(0)
  wait(getKey()==-1)

  if TxtFile:b7Axis or TxtFile:b8Axis
    call UI:Control_PanelMd("外部轴在运动")
  endIf

  if DataBase:bExtraContrAxis

    call UI:Control_PanelMd("等待PLC控制外部轴到位")
  endIf



  // wait(Motion:bMoveTask)
  wait(DataBase:nPointType>0)
  //轮询
  while DataBase:bMoveTask
    //强制使用离散工艺
    TxtFile:bMatchPreset=false

    if nPointType!=DataBase:nPointType

      l_nPointIndex=0
      n500Count=0
      nPointType=DataBase:nPointType
      //获取内容
      call GetListItems()
      cls()
      switch DataBase:nPointType
        case 1
          l_sItemTitle="趋近点"
          call UI:Control_Mess("类型:"+TxtFile:sTrajType[TxtFile:nSingleType],"趋近点个数:"+toString("",size(TxtFile:pAppro)))
        break

        case 2
          l_sItemTitle="切割点"
          if x_nTrajIndex<0
            call UI:Control_Mess("类型:"+TxtFile:sTrajType[TxtFile:nSingleType],"切割点个数:"+toString("",size(TxtFile:pCut)))
          else
            call UI:Control_Mess("类型:"+TxtFile:sTrajType[TxtFile:nSingleType],"切割点个数:"+toString("",TxtFile:trPointCount.y))
          endIf
        break
        case 3
          l_sItemTitle="离开点"
          call UI:Control_Mess("类型:"+TxtFile:sTrajType[TxtFile:nSingleType],"离开点个数:"+toString("",size(TxtFile:pLeave)))
        break
      endSwitch
    endIf



    l_nKey=getKey()
    switch l_nKey

      //激光
      case 271
        l_bKeyIO[0]=!l_bKeyIO[0]
        if l_bKeyIO[0]
          l_bKeyIO[2]=true
        endIf
      break

      //随动
      case 272
        l_bKeyIO[1]=!l_bKeyIO[1]
      break

      //气体
      case 273
        if !l_bKeyIO[0]
          l_bKeyIO[2]=!l_bKeyIO[2]
        else
          l_bKeyIO[2]=true
        endIf
      break

      //退出
      case 278
        call UI:Control_YesNO("确定要终止模拟吗?",l_bRes)
        if l_bRes
          DataBase:bMoveTask=false
          DataBase:bStopSimul=true
          taskKill("Simulation")
          wait(taskStatus("Simulation")==-1)
          //Motion:
          call Motion:KillTask()
          resetMotion()
          disablePower()
          call IO:SafteyIO()
          return
        endIf
      break




    endSwitch


    DataBase:nID=getMoveId()
    if ((DataBase:nID%500)>(l_nPointIndex+0.8)) or l_nKey!=-1 or DataBase:bPowerOn!=isPowered() or l_nPointIndex>(DataBase:nID%500-0.7) or l_nPointIndex<=0

      DataBase:bPowerOn=isPowered()
      //没有上电
      if !DataBase:bPowerOn
        l_bKeyIO[0]=l_bKeyIO[1]=l_bKeyIO[2]=false
      else
        //在切割点的时候
        if DataBase:nPointType==2
          //对于IO进行赋值
          //

          //          if !TxtFile:bWeldEnable
          //
          //            call IO:KeyDigtalIO(l_bKeyIO[2],l_bKeyIO[1],l_bKeyIO[0],TxtFile:trIODelay.x,TxtFile:trIODelay.y)
          //           // DataBase:bSimuIO=true
          //          else

          //2015.02.03
          if DataBase:bIOStart and TxtFile:trWorkplace.rz!=-1
            if !TxtFile:bWeldEnable or (TxtFile:bWeldEnable and !(TxtFile:trWorkplace.z==1))
              call IO:KeyDigtalIO(l_bKeyIO[2],l_bKeyIO[1],l_bKeyIO[0],TxtFile:trIODelay.x,TxtFile:trIODelay.y)
              // DataBase:bSimuIO=true
            endIf
          endIf

          //
          //          endIf
          if roundDown(DataBase:nID/500)!=n500Count
            n500Count=roundDown(DataBase:nID/500)
            call GetListItems()
          endIf

          // else
          // call IO:KeyDigtalIO(false,false,false,0,0)
          // DataBase:bSimuIO=false
        endIf

        //点序号变化
        // l_nPointIndex=max((round(DataBase:nID))%500-1,0)
        if (DataBase:nID-roundDown(DataBase:nID))>0.8
          l_nPointIndex=max(roundUp((DataBase:nID))%500-1,0)
        else
          l_nPointIndex=max(roundDown(DataBase:nID)%500-1,0)
        endIf



        //使用动作
        if TxtFile:bWeldEnable and TxtFile:trWorkplace.z==1

          call IO:GetKeyIO(l_bKeyIO[0],l_bKeyIO[1],l_bKeyIO[2])
        endIf

        switch DataBase:nPointType
          case 1
            l_nPointIndex=min(l_nPointIndex,size(TxtFile:pAppro)-1)
          break

          case 2
            l_nPointIndex=min(l_nPointIndex,size(TxtFile:pCut)-1)
          break


          case 3
            l_nPointIndex=min(l_nPointIndex,size(TxtFile:pLeave)-1)
          break
        endSwitch

      endIf
      //2016.04.07
      //模拟时候添加
     // if !TxtFile:bWeldEnable
        if false
        call UI:Form_Simulation("LasMAN3.6->模拟路径"+toString("",DataBase:nTrajIndex),l_sItemTitle,sSItem,l_nPointIndex,DataBase:nPresetData,l_bKeyIO)
      else
        l_trArray=TxtFile:trArray
        l_trArray.y=DataBase:nArrayX
        l_trArray.rx=DataBase:nArrayY
        l_trArray.rz=DataBase:nArrayZ

        call UI:Form_SimArray("LasMAN3.6->模拟路径"+toString("",DataBase:nTrajIndex),l_sItemTitle,sSItem,l_nPointIndex,DataBase:nPresetData,l_bKeyIO,l_trArray)
      endIf




      //2015.02.03 为同步轴设置
      if TxtFile:trWorkplace.rz==-1
        gotoxy(0,12)
        put("(穿孔工艺-1,空走)")
      endIf
      //

    endIf
    //2014.4.28
    DataBase:bKeyIO[0]=l_bKeyIO[0]
    DataBase:bKeyIO[1]=l_bKeyIO[1]
    DataBase:bKeyIO[2]=l_bKeyIO[2]

    delay(0)
  endWhile


  cls()

  //2014.3.6
  //模拟时初始化
  TxtFile:bStartRead=false

  //  if isEmpty() and taskStatus("Simulation")==-1
  //
  //    //call UI:Control_PanelMd("模拟成功")
  //   // delay(3)
  //    cls()
  //    return
  //  endIf
  //



end

--- SingleMove.pgx ---
program SingleMove(num x_nType)
  local bool l_bRes
  local jointRx l_jBuff
  local point l_p
begin
  //判断单个点是否可达



  resetMotion()
  setTextMode(0)
  gotoxy(0,0)
  put("                     ")

  //  //2014.07.28
  //  //同步七八轴
  //  if TxtFile:bSync7Axis or TxtFile:bSync8Axis
  //    if !ExtAxis:libExist("Disk://extAxisCan/extAxisCan.pjx")
  //      if ExtAxis:libLoad("Disk://extAxisCan/extAxisCan.pjx")!=0
  //        popUpMsg("加载外部轴出错")
  //        disablePower()
  //        DataBase:nPointType=5
  //        return
  //      endIf
  //    endIf
  //  endIf

  //2014.07.28
  //同步轴选项

  //2015.04.21
  //
  if TxtFile:nSingleType==20 or TxtFile:nSingleType==9
    if TxtFile:bSync7Axis==false and TxtFile:bSync8Axis==false
      popUpMsg("请先配置同步轴!")
      disablePower()
      DataBase:nPointType=5
      DataBase:bMoveTask=false
      return
    endIf
  endIf



  //*************************************
  //2014.12.08
  //修改基于第七轴坐标系点的判断
  if (TxtFile:nSingleType==20 or TxtFile:nSingleType==9)
    //and ExtAxis:bMoveType

    switch x_nType
      case 1
        call Motion:SpeedFilter(TxtFile:trAppro[nApproIndex],mNomSpeed)
        mNomSpeed.blend=off
        if TxtFile:bAppro[nApproIndex]

          call ExtAxis:SingleMove(2,l_jBuff,l_p,TxtFile:pAppro[nApproIndex],TxtFile:tCfg,mNomSpeed,TxtFile:trApproAxis[nApproIndex])
        else
          call ExtAxis:SingleMove(1,TxtFile:jAppro[nApproIndex],l_p,TxtFile:pAppro[nApproIndex],TxtFile:tCfg,mNomSpeed,TxtFile:trApproAxis[nApproIndex])
        endIf
      break


      case 2
        call Motion:SpeedFilter(TxtFile:trCut[nCutIndex],mNomSpeed)
        mNomSpeed.blend=off
        if TxtFile:bMoveC[nCutIndex] and nCutMc==0
          if TxtFile:pMoveC[nCutIndex]!=TxtFile:pCut[nCutIndex]
            call ExtAxis:SingleMove(3,l_jBuff,TxtFile:pMoveC[nCutIndex],TxtFile:pCut[nCutIndex],TxtFile:tCfg,mNomSpeed,TxtFile:trCutAxis[nCutIndex])
          endIf
        else
          if  TxtFile:bMoveC[nCutIndex] and nCutMc==1
            call ExtAxis:SingleMove(2,l_jBuff,l_p,TxtFile:pMoveC[nCutIndex],TxtFile:tCfg,mNomSpeed,TxtFile:trCutAxis[nCutIndex])
          else
            call ExtAxis:SingleMove(2,l_jBuff,l_p,TxtFile:pCut[nCutIndex],TxtFile:tCfg,mNomSpeed,TxtFile:trCutAxis[nCutIndex])
          endIf
        endIf
      break




      case 3
        call Motion:SpeedFilter(TxtFile:trLeave[nLeaveIndex],mNomSpeed)
        mNomSpeed.blend=off
        if TxtFile:bLeave[nLeaveIndex]
          call ExtAxis:SingleMove(2,l_jBuff,l_p,TxtFile:pLeave[nLeaveIndex],TxtFile:tCfg,mNomSpeed,TxtFile:trLeaveAxis[nLeaveIndex])
        else
          call ExtAxis:SingleMove(1,TxtFile:jLeave[nLeaveIndex],l_p,TxtFile:pLeave[nLeaveIndex],TxtFile:tCfg,mNomSpeed,TxtFile:trLeaveAxis[nLeaveIndex])
        endIf
      break

    endSwitch
    //2015.04.23
    //强制让其跳出
    return
  endIf



  //**********************************************
  //*************************************************


  switch x_nType


    //趋近点
    case 1

      call Motion:SpeedFilter(TxtFile:trAppro[nApproIndex],mNomSpeed)
      mNomSpeed.blend=off
      if TxtFile:bAppro[nApproIndex]
        call IsPointOK(nApproIndex,1,nCutMc,l_bRes)
        if l_bRes
          if TxtFile:nSingleType!=20 and TxtFile:nSingleType!=9
            movel(TxtFile:pAppro[nApproIndex],TxtFile:tCfg,mNomSpeed)
          else
            call ExtAxis:SingleMove(2,l_jBuff,l_p,TxtFile:pAppro[nApproIndex],TxtFile:tCfg,mNomSpeed,TxtFile:trApproAxis[nApproIndex])
          endIf
        else
          setTextMode(3)
          gotoxy(0,0)
          put("当前位置不可到达目标点")
        endIf
      else
        call Motion:Joint2Joint(TxtFile:jAppro[nApproIndex],l_jBuff,l_bRes)
        if !l_bRes
          popUpMsg("关节点转换出现异常")
          //return
        else
          //movej(l_jBuff,TxtFile:tCfg,mNomSpeed)

          if TxtFile:nSingleType!=20 and TxtFile:nSingleType!=9
            movej(l_jBuff,TxtFile:tCfg,mNomSpeed)
          else
            call ExtAxis:SingleMove(1,l_jBuff,l_p,TxtFile:pAppro[nApproIndex],TxtFile:tCfg,mNomSpeed,TxtFile:trApproAxis[nApproIndex])
          endIf



        endIf
      endIf



    break


    //切割点
    case 2
      //运动初始化
      if nCutIndex>=size(TxtFile:trCut)
        popUpMsg("nCutIndex序号异常")
      else
        call Motion:SpeedFilter(TxtFile:trCut[nCutIndex],mNomSpeed)
        mNomSpeed.blend=off
        call IsPointOK(nCutIndex,2,nCutMc,l_bRes)


        if l_bRes
          if TxtFile:bMoveC[nCutIndex] and nCutMc==0
            //2014.07.24
            //逆着走
            if nCutIndex<nCursonIndex
              if TxtFile:nSingleType!=20 and TxtFile:nSingleType!=9
                movel(TxtFile:pCut[nCutIndex],TxtFile:tCfg,mNomSpeed)
                movec(TxtFile:pMoveC[nCutIndex],TxtFile:pCut[nCutIndex-1],TxtFile:tCfg,mNomSpeed)
              else
                call ExtAxis:SingleMove(2,l_jBuff,l_p,TxtFile:pCut[nCutIndex],TxtFile:tCfg,mNomSpeed,TxtFile:trCutAxis[nCutIndex])
                call ExtAxis:SingleMove(3,l_jBuff,TxtFile:pMoveC[nCutIndex],TxtFile:pCut[nCutIndex-1],TxtFile:tCfg,mNomSpeed,TxtFile:trCutAxis[nCutIndex])

              endIf
            else
              if TxtFile:nSingleType!=20 and TxtFile:nSingleType!=9
                movel(TxtFile:pCut[nCutIndex-1],TxtFile:tCfg,mNomSpeed)
                movec(TxtFile:pMoveC[nCutIndex],TxtFile:pCut[nCutIndex],TxtFile:tCfg,mNomSpeed)
              else
                call ExtAxis:SingleMove(2,l_jBuff,l_p,TxtFile:pCut[nCutIndex-1],TxtFile:tCfg,mNomSpeed,TxtFile:trCutAxis[nCutIndex])
                call ExtAxis:SingleMove(3,l_jBuff,TxtFile:pMoveC[nCutIndex],TxtFile:pCut[nCutIndex],TxtFile:tCfg,mNomSpeed,TxtFile:trCutAxis[nCutIndex])
              endIf
            endIf

          else
            if TxtFile:bMoveC[nCutIndex] and nCutMc==1
              movel(TxtFile:pMoveC[nCutIndex],TxtFile:tCfg,mNomSpeed)
            else
              if TxtFile:nSingleType!=20 and TxtFile:nSingleType!=9
                movel(TxtFile:pCut[nCutIndex],TxtFile:tCfg,mNomSpeed)
              else
                call ExtAxis:SingleMove(2,l_jBuff,l_p,TxtFile:pCut[nCutIndex],TxtFile:tCfg,mNomSpeed,TxtFile:trCutAxis[nCutIndex])
              endIf
            endIf
          endIf

        else
          setTextMode(3)
          gotoxy(0,0)
          put("当前位置不可到达目标点")
        endIf


      endIf
    break




    //离开点
    case 3



      resetMotion()
      call Motion:SpeedFilter(TxtFile:trLeave[nLeaveIndex],mNomSpeed)
      mNomSpeed.blend=off

      if TxtFile:bLeave[nLeaveIndex]
        call IsPointOK(nLeaveIndex,3,nCutMc,l_bRes)
        if l_bRes
          //  movel(TxtFile:pLeave[nLeaveIndex],TxtFile:tCfg,mNomSpeed)
          if TxtFile:nSingleType!=20 and TxtFile:nSingleType!=9
            movel(TxtFile:pLeave[nLeaveIndex],TxtFile:tCfg,mNomSpeed)
          else
            call ExtAxis:SingleMove(2,l_jBuff,l_p,TxtFile:pLeave[nLeaveIndex],TxtFile:tCfg,mNomSpeed,TxtFile:trLeaveAxis[nLeaveIndex])
          endIf


        else
          setTextMode(3)
          gotoxy(0,0)
          put("当前位置不可到达目标点")
        endIf
      else
        call Motion:Joint2Joint(TxtFile:jLeave[nLeaveIndex],l_jBuff,l_bRes)
        if !l_bRes
          popUpMsg("关节点转换出现异常")
        else
          //  movej(l_jBuff,TxtFile:tCfg,mNomSpeed)

          if TxtFile:nSingleType!=20 and TxtFile:nSingleType!=9
            movej(l_jBuff,TxtFile:tCfg,mNomSpeed)
          else
            call ExtAxis:SingleMove(1,l_jBuff,l_p,TxtFile:pAppro[nApproIndex],TxtFile:tCfg,mNomSpeed,TxtFile:trLeaveAxis[nLeaveIndex])
          endIf



        endIf
      endIf


    break
  endSwitch


  setTextMode(0)






end

--- Teach2Tool.pgx ---
public program Teach2Tool()
  local point l_p[3]
  local num l_nIndex
  local num l_nKey
  local bool l_bRes
  local string l_sData[3]
  local tool l_tBuff
  local tool l_tTool
begin


  //使用拆工具法进行示教
  l_tBuff=TxtFile:tCfg
  link(l_p[0],world)
  link(l_p[1],world)
  link(l_p[2],world)
  link(l_tTool,flange)
  resetMotion()

  resize(sSItem,1,6)
  l_sData[0]="1.输入尖点值"
  l_sData[1]="2.示教装尖点点"
  l_sData[2]="3.示教带工具点"


  sSItem[0]="X   :"+toString(".3",l_tBuff.trsf.x)
  sSItem[1]="Y   :"+toString(".3",l_tBuff.trsf.y)
  sSItem[2]="Z   :"+toString(".3",l_tBuff.trsf.z)
  sSItem[3]="RX  :"+toString(".3",l_tBuff.trsf.rx)
  sSItem[4]="RY  :"+toString(".3",l_tBuff.trsf.ry)
  sSItem[5]="RZ  :"+toString(".3",l_tBuff.trsf.rz)



  cls()
  call UI:Form_LabelList("LasMAN3.6->示教工具","工具值",sSItem,"示教点",l_sData,l_nIndex,"记录,对齐,,,上传,计算,保存,退出")

  while  true
    l_nKey=getKey()
    switch l_nKey
      case 261
        l_nIndex=max(l_nIndex-1,0)

        resetMotion()
        mNomSpeed.blend=off

        switch l_nIndex
          case 1
            movej(l_p[1],l_tTool,mNomSpeed)
          break

          case 2
            movej(l_p[2],flange,mNomSpeed)
          break
        endSwitch

      break


      case 266
        l_nIndex=min(l_nIndex+1,2)
        resetMotion()
        mNomSpeed.blend=off
        switch l_nIndex
          case 1
            movej(l_p[1],l_tTool,mNomSpeed)
          break

          case 2
            movej(l_p[2],flange,mNomSpeed)
          break
        endSwitch
      break




      //记录
      case 271
        call UI:Control_YesNO("确定要记录吗?",l_bRes)
        l_tTool.trsf={0,0,0,0,0,0}
        l_tTool.trsf.z=l_p[0].trsf.z
        if l_bRes
          switch l_nIndex
            case 1
              l_p[1]=here(l_tTool,world)
            break

            case 2
              l_p[2]=here(flange,world)
            break
          endSwitch
        endIf
      break

      //对齐
      case 272
        call Kit:Align(l_tBuff)

      break


      //上传
      case 275
        call UI:Control_YesNO("确定要上传吗?",l_bRes)
        if l_bRes
          call Kit:UpLoad()
        endIf

      break


      //计算
      case 276
        call UI:Control_YesNO("确定要计算吗?",l_bRes)
        if l_bRes
          l_tBuff.trsf=!l_p[2].trsf*l_p[1].trsf

          sSItem[0]="X   :"+toString(".3",l_tBuff.trsf.x)
          sSItem[1]="Y   :"+toString(".3",l_tBuff.trsf.y)
          sSItem[2]="Z   :"+toString(".3",l_tBuff.trsf.z)
          sSItem[3]="RX  :"+toString(".3",l_tBuff.trsf.rx)
          sSItem[4]="RY  :"+toString(".3",l_tBuff.trsf.ry)
          sSItem[5]="RZ  :"+toString(".3",l_tBuff.trsf.rz)
        endIf
      break



      //保存
      case 277
        call UI:Control_YesNO("确定要保存吗?",l_bRes)
        if l_bRes

          TxtFile:tCfg.trsf=l_tBuff.trsf
          call TxtFile:SaveCfg(l_bRes)
          if !l_bRes
            popUpMsg("保存错误")
          else
            popUpMsg("保存成功")
          endIf
        endIf



      break




      //退出
      case 278
        call UI:Control_YesNO("确定要退出吗?",l_bRes)
        if l_bRes

          return
        endIf
      break

      //点位
      case 270
        call UI:Control_Point(l_p[l_nIndex])
        if l_nIndex==0
          l_p[0].trsf={0,0,l_p[0].trsf.z,0,0,0}
        endIf
      break

    endSwitch

    if l_nKey!=-1
      call UI:Form_LabelList("LasMAN3.6->示教工具","工具值",sSItem,"参考点",l_sData,l_nIndex,"记录,对齐,,,上传,计算,保存,退出")

    endIf

    delay(0)

  endWhile







end

--- TeachAction.pgx ---
public program TeachAction()
  local num l_nKey
  local num l_nPointType
  local num l_nPointIndex
  local bool l_bRes
  local string l_sItemTitle
  local bool l_bKeyIO
  local num l_nNum
  local string l_sBuff[8]
  local num l_nIOSeq
begin

  //动作示教
  //参数初始化

  resetMotion()
  userPage()
  DataBase:bStopPoll=true

  call TxtFile:ReadAction(l_bRes)
  if !l_bRes
    popUpMsg("读取动作文件不正确")
    return
  endIf

  //轮询
  resize(sSItem,1,50)
  for l_nNum=0 to 49
    sSItem[l_nNum]="序号:"+toString("",l_nNum+1)

  endFor
  for l_nNum=0 to 3
    l_sBuff[2*l_nNum+0]=IO:sIOName[TxtFile:nAction[l_nPointIndex+1,l_nNum+l_nIOSeq*4,0]]
    l_sBuff[2*l_nNum+0]=toString("",l_nNum+l_nIOSeq*4+1)+"名称:"+ l_sBuff[2*l_nNum+0]
    l_sBuff[2*l_nNum+1]="值:"+toString(".3",TxtFile:nAction[l_nPointIndex+1,l_nNum+l_nIOSeq*4,1])

  endFor
  cls()
  call UI:Form_Action("LasMAN3.6->示教动作","动作表",sSItem,l_nPointIndex,l_bKeyIO,l_nPointIndex+1,l_sBuff)



  DataBase:bStopPoll=false

  while true

    l_nKey=getKey()
    switch l_nKey

      //执行
      case 271
        nTeachAction=l_nPointIndex+1
        l_bKeyIO[0]=!l_bKeyIO[0]
        if l_bKeyIO
          if !isPowered()
            popUpMsg("请先上电")
            l_bKeyIO=!l_bKeyIO
          else
            taskCreate "Action",100, OnAction()
          endIf
        else
          if taskStatus("Action")!=-1
            taskKill("Action")

          endIf


        endIf
      break


      //上传
      case 275
        call UI:Control_YesNO("确定要上传吗?",l_bRes)
        if l_bRes
          call Kit:UpLoad()
          //return
        endIf
      break


      //退出
      case 278
        call UI:Control_YesNO("确定要退出吗?",l_bRes)
        if l_bRes
          if taskStatus("Action")!=-1
            taskKill("Action")

          endIf
          return
        endIf
      break


      //修改
      case 276,270
        if l_bKeyIO
          popUpMsg("动作正在执行")
        else
          call UI:Control_Action(TxtFile:nAction,l_nPointIndex+1,IO:sIOName,IO:bDigtal)
        endIf
        cls()
      break


      case 277
        call UI:Control_YesNO("确定要保存吗?",l_bRes)
        if l_bRes
          call TxtFile:SaveAction(l_bRes)
          if !l_bRes
            popUpMsg("保存出错")
          else
            popUpMsg("保存成功")
          endIf
          cls()
          // return
        endIf
      break

      case 264
        l_nIOSeq=max(0,l_nIOSeq-1)

      break


      case 268
        l_nIOSeq=min(2,l_nIOSeq+1)

      break


      case 261
        l_nPointIndex=max(0,l_nPointIndex-1)
        l_nIOSeq=0
         disablePower()
      break


      case 266
        l_nPointIndex=min(size(sSItem)-1,l_nPointIndex+1)
        l_nIOSeq=0
         disablePower()
      break




    endSwitch

    if !DataBase:bPowerOn
      l_bKeyIO=false
      if taskStatus("Action")!=-1
        taskKill("Action")
        wait(taskStatus("Action")==-1)
      endIf
    endIf
    if l_nKey!=-1  and l_nKey>=260
      for l_nNum=0 to 3

        l_sBuff[2*l_nNum+0]=IO:sIOName[TxtFile:nAction[l_nPointIndex+1,l_nNum+l_nIOSeq*4,0]]
        l_sBuff[2*l_nNum+0]=toString("",l_nNum+l_nIOSeq*4+1)+"名称:"+ l_sBuff[2*l_nNum+0]
        l_sBuff[2*l_nNum+1]="值:"+toString(".3",TxtFile:nAction[l_nPointIndex+1,l_nNum+l_nIOSeq*4,1])


      endFor
      call UI:Form_Action("LasMAN3.6->示教动作","动作表",sSItem,l_nPointIndex,l_bKeyIO,l_nPointIndex+1,l_sBuff)


    endIf




  endWhile









end

--- TeachAxis.pgx ---
public program TeachAxis(num& x_nPosition, num& x_nSpeed, num& x_nPrecent, num& x_nJogSpeed, bool x_b8Axis)
  local num l_nKey
  local bool l_bRes
  local num l_nIndex
  local num l_nSpeed
  local num l_nPosition
  local bool l_bFirst
  local bool l_bPowerOn
  local bool l_bAlarm
  local num l_nPrecent
  local num l_nJogSpeed
  local bool l_bBHome
  local num l_nBuff
  local string l_sBottom
begin
  //七轴示教
  resetMotion()

  wait(isKeyPressed(272)==false)


  resize(sSItem,1,7)
  //  sSItem[0]="参数"
  //  sSItem[1]="复位"

  l_nPosition=x_nPosition
  l_nSpeed=x_nSpeed
  l_nPrecent=x_nPrecent
  l_nJogSpeed=x_nJogSpeed
  cls()
  //  call UI:Form_PanelList("LasMAN3.6->示教异步七轴","第七轴",sSItem,l_nIndex,"+,-,记录,回零,运动,停止,保存,退出")
  //  call UI:Control_Mess("马达正常,未上电","")

  if DataBase:nInterfaceType==12 or DataBase:nInterfaceType==16
    bCheckAxisSafte=false

  endIf
  call UI:Control_PanelMd("等待外部轴安全门打开")
  call IO:AxisJogSpeed(l_nJogSpeed,x_b8Axis)

  call IO:AxisDoor(true,x_b8Axis)
  cls()
  while  DataBase:nInterfaceType==12 or DataBase:nInterfaceType==5 or DataBase:nInterfaceType==16
    //
    if !x_b8Axis
      call IO:Axis7Status(l_bPowerOn,l_bAlarm,l_bBHome)
    else
      call IO:Axis8Status(l_bPowerOn,l_bAlarm,l_bBHome)
    endIf

    //判断按键是否一直按着
    l_nKey=getKey()
    if isKeyPressed(271)
      l_nKey=271
    endIf

    if isKeyPressed(272)
      l_nKey=272
    endIf


    switch l_nKey
      //回零测试

      case 97
        call IO:AxisTest()
      break


      //复位
      //      case 113
      //        call UI:Control_YesNO("确定需要复位吗？",l_bRes)
      //        if l_bRes
      //          if x_b8Axis
      //            call IO:Axis8Action(10)
      //          else
      //            call IO:Axis7Action(10)
      //          endIf
      //        endIf
      //      break

      //向上
      case 261
        l_nIndex=max(0,l_nIndex-1)

      break

      //向下
      case 266
        l_nIndex=min(6,l_nIndex+1)
      break


      //+
      case 271
        if l_bAlarm
          popUpMsg("马达报警，请先复位")

        else
          if !isPowered()
            popUpMsg("请先上电")
          else
            if x_b8Axis
              call IO:Axis8Action(1)
            else
              call IO:Axis7Action(1)
            endIf
          endIf
        endIf
      break


      //-
      case 272
        if l_bAlarm
          popUpMsg("马达报警，请先复位")

        else
          if !isPowered()
            popUpMsg("请先上电")
          else
            if x_b8Axis
              call IO:Axis8Action(2)
            else
              call IO:Axis7Action(2)
            endIf
          endIf
        endIf
      break





      //记录
      case 273
        if !l_bBHome
          popUpMsg("请先回零")

        else
          call IO:AxisIsNeg(x_b8Axis,l_bRes)
          if l_bRes
            popUpMsg("数值过大或为负,请点动+到正值")
          else
            if !bCheckAxisSafte
              call UI:Control_YesNO("确定需要记录吗？",l_bRes)
              if l_bRes
                if !x_b8Axis
                  call IO:GetAxis7Pos(l_nPosition,l_nPrecent)
                  //TxtFile:trAxisData.y=l_nSpeed
                else
                  call IO:GetAxis8Pos(l_nPosition,l_nPrecent)
                  // TxtFile:trAxis8Data.y=l_nSpeed
                endIf
              endIf
            endIf
          endIf
        endIf
      break


      //回零
      case 274
        if isPowered()
          if l_bAlarm
            popUpMsg("马达报警，请先复位")
          else
            call UI:Control_YesNO("确定需要回机械原点吗？",l_bRes)
            if l_bRes
              call UI:Control_PanelMd("异步外部轴马达正在回机械零位")
              if !x_b8Axis
                call IO:Axis7Action(4)
              else
                call IO:Axis8Action(4)
              endIf
              cls()
            endIf
          endIf
        else
          popUpMsg("机械手臂先上电")
        endIf
      break




      //运动
      case 275
        if isPowered()
          if l_bAlarm
            popUpMsg("马达报警，请先复位")

          else
            if !l_bBHome
              popUpMsg("请先回到机械零位哦")
            else
              call UI:Control_YesNO("确定需要运动吗？",l_bRes)
              if l_bRes
                call UI:Control_PanelMd("异步外部轴马达正在运动")
                if !x_b8Axis
                  call IO:Axis7OnReady(l_nPosition,l_nSpeed,l_nPrecent,l_bRes)
                else
                  call IO:Axis8OnReady(l_nPosition,l_nSpeed,l_nPrecent,l_bRes)
                endIf
                cls()
                if l_bRes
                  popUpMsg("运动到位")
                else
                  popUpMsg("运动出错")
                endIf

              endIf
            endIf
          endIf
        else

          popUpMsg("机械手臂先上电")
        endIf

      break






      //停止
      case 276
        if DataBase:nInterfaceType!=5
          call UI:Control_YesNO("确定需要上传吗？",l_bRes)
          if l_bRes
            //            if x_b8Axis
            //              call IO:Axis8Action(6)
            //            else
            //              call IO:Axis7Action(6)
            //            endIf
            //          endIf
            call Kit:UpLoad()
          endIf
        endIf

      break


      //保存
      case 277
        if !bCheckAxisSafte
          call UI:Control_YesNO("确定需要保存吗？",l_bRes)
          if l_bRes
            x_nPosition=l_nPosition
            x_nSpeed=l_nSpeed
            x_nPrecent=l_nPrecent
            x_nJogSpeed=l_nJogSpeed
            nAxisSpeed=l_nSpeed
            //生产配置文件
            if DataBase:nInterfaceType!=5
              call TxtFile:SaveCfg(l_bRes)
            endIf


            if l_bRes
              popUpMsg("保存成功")
            else
              popUpMsg("保存失败")
            endIf

          endIf
        endIf
      break

      //
      case 278,255
        if x_nPosition!=l_nPosition or  x_nSpeed != l_nSpeed or x_nPrecent!=l_nPrecent
          call UI:Control_YesNO("参数未保存,确定需要退出吗？",l_bRes)
          if l_bRes
            cls()
            return
          endIf
        else
          cls()
          return
        endIf

      break


      case 270

        switch l_nIndex

          case 0,1,2,3
            if !bCheckAxisSafte
              call UI:Control_AxisPar(l_nPosition,l_nSpeed,l_nPrecent,l_nJogSpeed,DataBase:nInterfaceType==5)
              call IO:AxisJogSpeed(l_nJogSpeed,x_b8Axis)
            endIf
          break

          case 4
            call UI:Control_YesNO("确定需要复位吗？",l_bRes)
            if l_bRes
              if x_b8Axis
                call IO:Axis8Action(10)
              else
                call IO:Axis7Action(10)
              endIf
            endIf
          break

          case 5
            call UI:Control_YesNO("确定需要开门吗？",l_bRes)
            if l_bRes
              call UI:Control_PanelMd("正在打开门....")
              if x_b8Axis
                call IO:AxisDoor(true,true)
              else
                call IO:AxisDoor(true,false)
              endIf
              cls()
            endIf
          break


